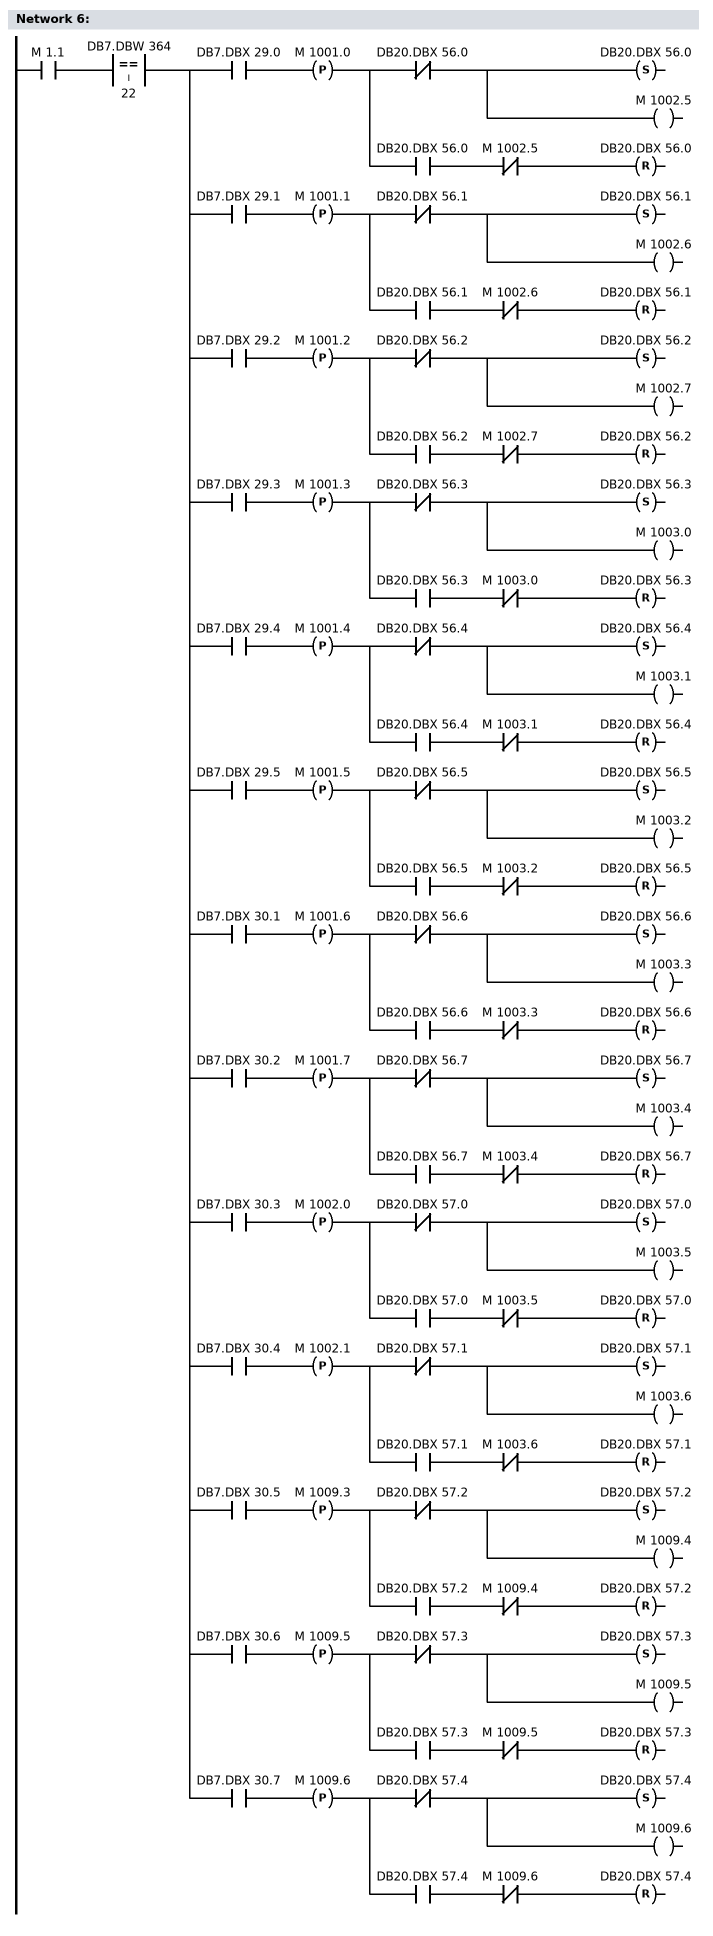
NETWORK
TITLE =
      A     M 1.1;
      A(;
      L     DB7.DBW 364;
      L     22;
      ==I;
      );
      =     L 0.0;
      A     L 0.0;
      A     DB7.DBX 29.0;
      FP    M 1001.0;
      =     L 0.1;
      A     L 0.1;
      AN    DB20.DBX 56.0;
      S     DB20.DBX 56.0;
      =     M 1002.5;
      A     L 0.1;
      A     DB20.DBX 56.0;
      AN    M 1002.5;
      R     DB20.DBX 56.0;
      A     L 0.0;
      A     DB7.DBX 29.1;
      FP    M 1001.1;
      =     L 0.1;
      A     L 0.1;
      AN    DB20.DBX 56.1;
      S     DB20.DBX 56.1;
      =     M 1002.6;
      A     L 0.1;
      A     DB20.DBX 56.1;
      AN    M 1002.6;
      R     DB20.DBX 56.1;
      A     L 0.0;
      A     DB7.DBX 29.2;
      FP    M 1001.2;
      =     L 0.1;
      A     L 0.1;
      AN    DB20.DBX 56.2;
      S     DB20.DBX 56.2;
      =     M 1002.7;
      A     L 0.1;
      A     DB20.DBX 56.2;
      AN    M 1002.7;
      R     DB20.DBX 56.2;
      A     L 0.0;
      A     DB7.DBX 29.3;
      FP    M 1001.3;
      =     L 0.1;
      A     L 0.1;
      AN    DB20.DBX 56.3;
      S     DB20.DBX 56.3;
      =     M 1003.0;
      A     L 0.1;
      A     DB20.DBX 56.3;
      AN    M 1003.0;
      R     DB20.DBX 56.3;
      A     L 0.0;
      A     DB7.DBX 29.4;
      FP    M 1001.4;
      =     L 0.1;
      A     L 0.1;
      AN    DB20.DBX 56.4;
      S     DB20.DBX 56.4;
      =     M 1003.1;
      A     L 0.1;
      A     DB20.DBX 56.4;
      AN    M 1003.1;
      R     DB20.DBX 56.4;
      A     L 0.0;
      A     DB7.DBX 29.5;
      FP    M 1001.5;
      =     L 0.1;
      A     L 0.1;
      AN    DB20.DBX 56.5;
      S     DB20.DBX 56.5;
      =     M 1003.2;
      A     L 0.1;
      A     DB20.DBX 56.5;
      AN    M 1003.2;
      R     DB20.DBX 56.5;
      A     L 0.0;
      A     DB7.DBX 30.1;
      FP    M 1001.6;
      =     L 0.1;
      A     L 0.1;
      AN    DB20.DBX 56.6;
      S     DB20.DBX 56.6;
      =     M 1003.3;
      A     L 0.1;
      A     DB20.DBX 56.6;
      AN    M 1003.3;
      R     DB20.DBX 56.6;
      A     L 0.0;
      A     DB7.DBX 30.2;
      FP    M 1001.7;
      =     L 0.1;
      A     L 0.1;
      AN    DB20.DBX 56.7;
      S     DB20.DBX 56.7;
      =     M 1003.4;
      A     L 0.1;
      A     DB20.DBX 56.7;
      AN    M 1003.4;
      R     DB20.DBX 56.7;
      A     L 0.0;
      A     DB7.DBX 30.3;
      FP    M 1002.0;
      =     L 0.1;
      A     L 0.1;
      AN    DB20.DBX 57.0;
      S     DB20.DBX 57.0;
      =     M 1003.5;
      A     L 0.1;
      A     DB20.DBX 57.0;
      AN    M 1003.5;
      R     DB20.DBX 57.0;
      A     L 0.0;
      A     DB7.DBX 30.4;
      FP    M 1002.1;
      =     L 0.1;
      A     L 0.1;
      AN    DB20.DBX 57.1;
      S     DB20.DBX 57.1;
      =     M 1003.6;
      A     L 0.1;
      A     DB20.DBX 57.1;
      AN    M 1003.6;
      R     DB20.DBX 57.1;
      A     L 0.0;
      A     DB7.DBX 30.5;
      FP    M 1009.3;
      =     L 0.1;
      A     L 0.1;
      AN    DB20.DBX 57.2;
      S     DB20.DBX 57.2;
      =     M 1009.4;
      A     L 0.1;
      A     DB20.DBX 57.2;
      AN    M 1009.4;
      R     DB20.DBX 57.2;
      A     L 0.0;
      A     DB7.DBX 30.6;
      FP    M 1009.5;
      =     L 0.1;
      A     L 0.1;
      AN    DB20.DBX 57.3;
      S     DB20.DBX 57.3;
      =     M 1009.5;
      A     L 0.1;
      A     DB20.DBX 57.3;
      AN    M 1009.5;
      R     DB20.DBX 57.3;
      A     L 0.0;
      A     DB7.DBX 30.7;
      FP    M 1009.6;
      =     L 0.1;
      A     L 0.1;
      AN    DB20.DBX 57.4;
      S     DB20.DBX 57.4;
      =     M 1009.6;
      A     L 0.1;
      A     DB20.DBX 57.4;
      AN    M 1009.6;
      R     DB20.DBX 57.4;
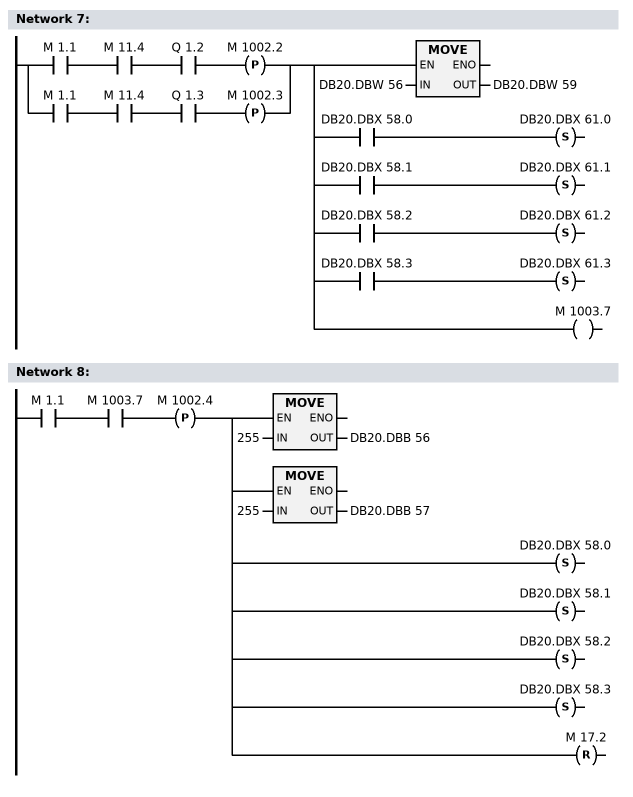
NETWORK
TITLE =
      A     M 1.1;
      A     M 11.4;
      A     Q 1.2;
      FP    M 1002.2;
      O(;
      A     M 1.1;
      A     M 11.4;
      A     Q 1.3;
      FP    M 1002.3;
      );
      =     L 0.0;
      A     L 0.0;
      JNB   M009;
      L     DB20.DBW 56;
      T     DB20.DBW 59;
M009: NOP   0;
      A     L 0.0;
      A     DB20.DBX 58.0;
      S     DB20.DBX 61.0;
      A     L 0.0;
      A     DB20.DBX 58.1;
      S     DB20.DBX 61.1;
      A     L 0.0;
      A     DB20.DBX 58.2;
      S     DB20.DBX 61.2;
      A     L 0.0;
      A     DB20.DBX 58.3;
      S     DB20.DBX 61.3;
      A     L 0.0;
      BLD   102;
      =     M 1003.7;
NETWORK
TITLE =
      A     M 1.1;
      A     M 1003.7;
      FP    M 1002.4;
      =     L 0.0;
      A     L 0.0;
      JNB   M010;
      L     255;
      T     DB20.DBB 56;
M010: NOP   0;
      A     L 0.0;
      JNB   M011;
      L     255;
      T     DB20.DBB 57;
M011: NOP   0;
      A     L 0.0;
      BLD   102;
      S     DB20.DBX 58.0;
      A     L 0.0;
      BLD   102;
      S     DB20.DBX 58.1;
      A     L 0.0;
      BLD   102;
      S     DB20.DBX 58.2;
      A     L 0.0;
      BLD   102;
      S     DB20.DBX 58.3;
      A     L 0.0;
      BLD   102;
      R     M 17.2;
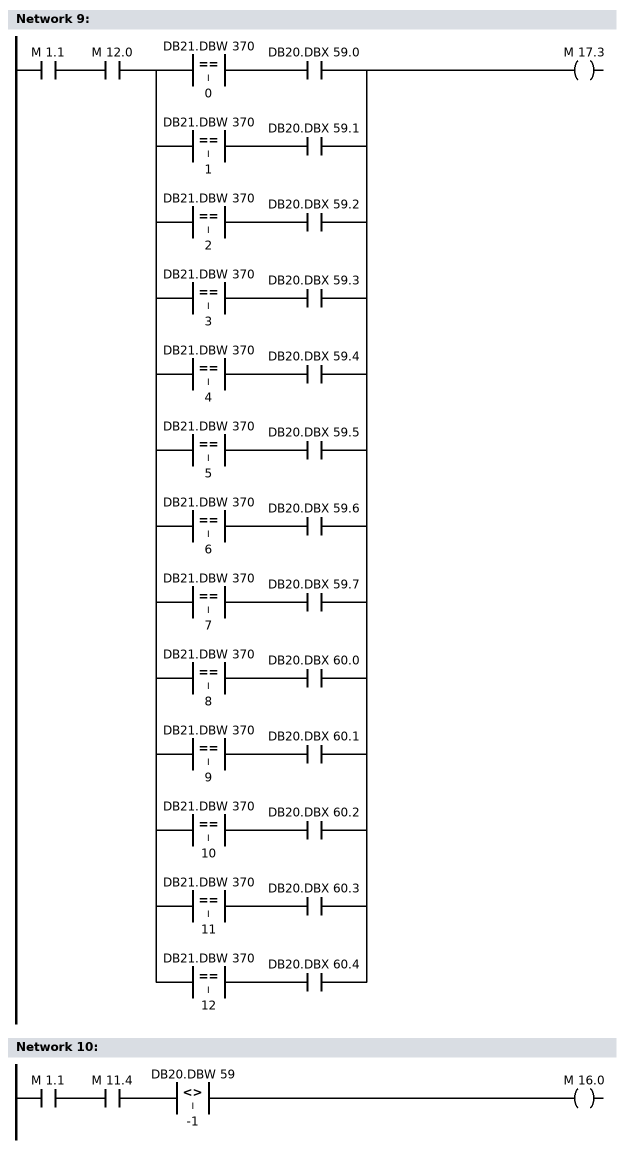
NETWORK
TITLE =
      A     M 1.1;
      A     M 12.0;
      A(;
      A(;
      L     DB21.DBW 370;
      L     0;
      ==I;
      );
      A     DB20.DBX 59.0;
      O;
      A(;
      L     DB21.DBW 370;
      L     1;
      ==I;
      );
      A     DB20.DBX 59.1;
      O;
      A(;
      L     DB21.DBW 370;
      L     2;
      ==I;
      );
      A     DB20.DBX 59.2;
      O;
      A(;
      L     DB21.DBW 370;
      L     3;
      ==I;
      );
      A     DB20.DBX 59.3;
      O;
      A(;
      L     DB21.DBW 370;
      L     4;
      ==I;
      );
      A     DB20.DBX 59.4;
      O;
      A(;
      L     DB21.DBW 370;
      L     5;
      ==I;
      );
      A     DB20.DBX 59.5;
      O;
      A(;
      L     DB21.DBW 370;
      L     6;
      ==I;
      );
      A     DB20.DBX 59.6;
      O;
      A(;
      L     DB21.DBW 370;
      L     7;
      ==I;
      );
      A     DB20.DBX 59.7;
      O;
      A(;
      L     DB21.DBW 370;
      L     8;
      ==I;
      );
      A     DB20.DBX 60.0;
      O;
      A(;
      L     DB21.DBW 370;
      L     9;
      ==I;
      );
      A     DB20.DBX 60.1;
      O;
      A(;
      L     DB21.DBW 370;
      L     10;
      ==I;
      );
      A     DB20.DBX 60.2;
      O;
      A(;
      L     DB21.DBW 370;
      L     11;
      ==I;
      );
      A     DB20.DBX 60.3;
      O;
      A(;
      L     DB21.DBW 370;
      L     12;
      ==I;
      );
      A     DB20.DBX 60.4;
      );
      =     M 17.3;
NETWORK
TITLE =
      A     M 1.1;
      A     M 11.4;
      A(;
      L     DB20.DBW 59;
      L     -1;
      <>I;
      );
      =     M 16.0;
END_FUNCTION

FUNCTION FC 54 : VOID
VERSION : 0.1
BEGIN
// (block stored without names or comments; labels and parameter names are numbered)
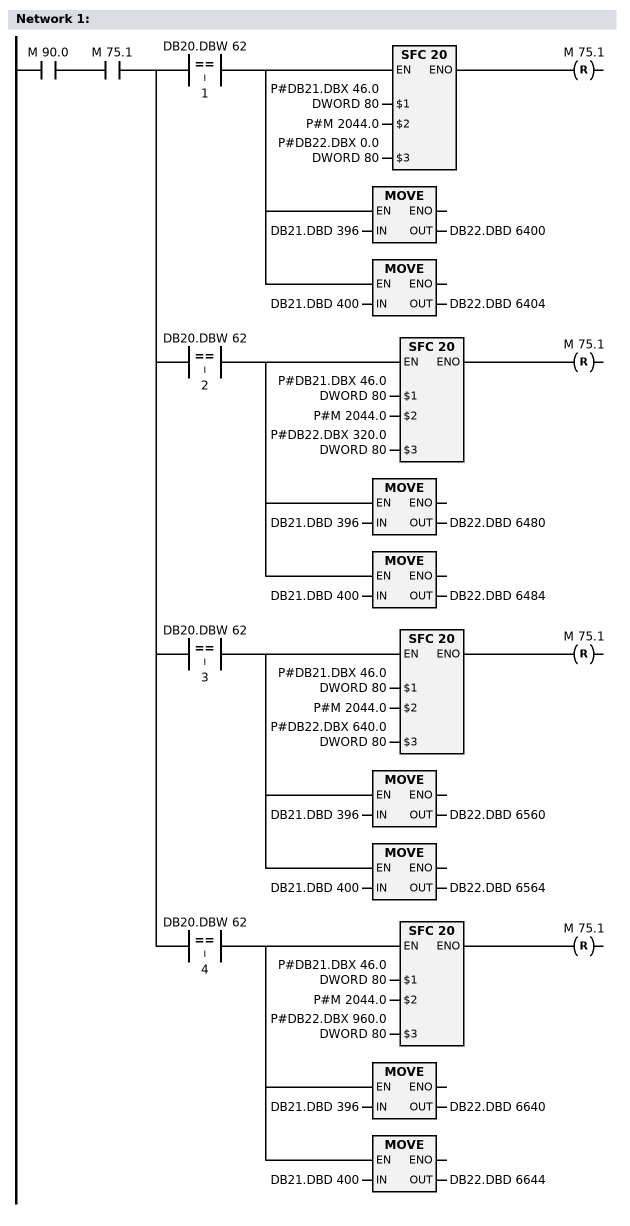
NETWORK
TITLE =
      A     M 90.0;
      A     M 75.1;
      =     L 0.0;
      A     L 0.0;
      A(;
      L     DB20.DBW 62;
      L     1;
      ==I;
      );
      =     L 0.1;
      A     L 0.1;
      JNB   M001;
      CALL  SFC 20 (
           $1                       := P#DB21.DBX 46.0 DWORD 80,
           $2                       := P#M 2044.0,
           $3                       := P#DB22.DBX 0.0 DWORD 80);
M001: A     BR;
      R     M 75.1;
      A     L 0.1;
      JNB   M002;
      L     DB21.DBD 396;
      T     DB22.DBD 6400;
M002: NOP   0;
      A     L 0.1;
      JNB   M003;
      L     DB21.DBD 400;
      T     DB22.DBD 6404;
M003: NOP   0;
      A     L 0.0;
      A(;
      L     DB20.DBW 62;
      L     2;
      ==I;
      );
      =     L 0.1;
      A     L 0.1;
      JNB   M004;
      CALL  SFC 20 (
           $1                       := P#DB21.DBX 46.0 DWORD 80,
           $2                       := P#M 2044.0,
           $3                       := P#DB22.DBX 320.0 DWORD 80);
M004: A     BR;
      R     M 75.1;
      A     L 0.1;
      JNB   M005;
      L     DB21.DBD 396;
      T     DB22.DBD 6480;
M005: NOP   0;
      A     L 0.1;
      JNB   M006;
      L     DB21.DBD 400;
      T     DB22.DBD 6484;
M006: NOP   0;
      A     L 0.0;
      A(;
      L     DB20.DBW 62;
      L     3;
      ==I;
      );
      =     L 0.1;
      A     L 0.1;
      JNB   M007;
      CALL  SFC 20 (
           $1                       := P#DB21.DBX 46.0 DWORD 80,
           $2                       := P#M 2044.0,
           $3                       := P#DB22.DBX 640.0 DWORD 80);
M007: A     BR;
      R     M 75.1;
      A     L 0.1;
      JNB   M008;
      L     DB21.DBD 396;
      T     DB22.DBD 6560;
M008: NOP   0;
      A     L 0.1;
      JNB   M009;
      L     DB21.DBD 400;
      T     DB22.DBD 6564;
M009: NOP   0;
      A     L 0.0;
      A(;
      L     DB20.DBW 62;
      L     4;
      ==I;
      );
      =     L 0.1;
      A     L 0.1;
      JNB   M010;
      CALL  SFC 20 (
           $1                       := P#DB21.DBX 46.0 DWORD 80,
           $2                       := P#M 2044.0,
           $3                       := P#DB22.DBX 960.0 DWORD 80);
M010: A     BR;
      R     M 75.1;
      A     L 0.1;
      JNB   M011;
      L     DB21.DBD 396;
      T     DB22.DBD 6640;
M011: NOP   0;
      A     L 0.1;
      JNB   M012;
      L     DB21.DBD 400;
      T     DB22.DBD 6644;
M012: NOP   0;
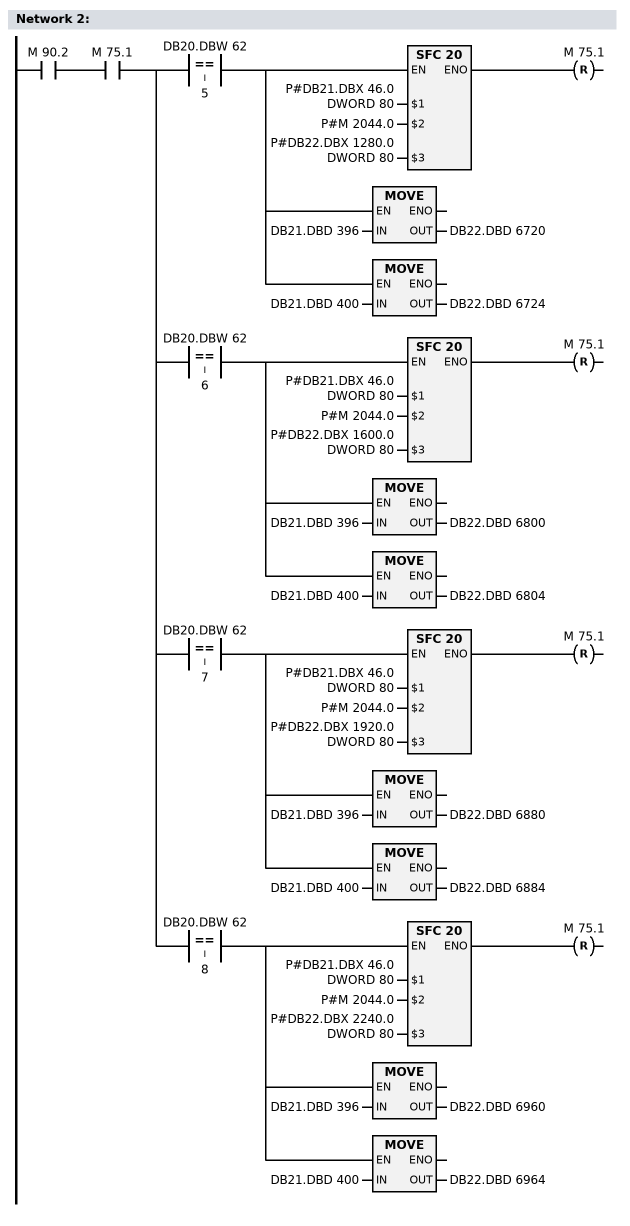
NETWORK
TITLE =
      A     M 90.2;
      A     M 75.1;
      =     L 0.0;
      A     L 0.0;
      A(;
      L     DB20.DBW 62;
      L     5;
      ==I;
      );
      =     L 0.1;
      A     L 0.1;
      JNB   M013;
      CALL  SFC 20 (
           $1                       := P#DB21.DBX 46.0 DWORD 80,
           $2                       := P#M 2044.0,
           $3                       := P#DB22.DBX 1280.0 DWORD 80);
M013: A     BR;
      R     M 75.1;
      A     L 0.1;
      JNB   M014;
      L     DB21.DBD 396;
      T     DB22.DBD 6720;
M014: NOP   0;
      A     L 0.1;
      JNB   M015;
      L     DB21.DBD 400;
      T     DB22.DBD 6724;
M015: NOP   0;
      A     L 0.0;
      A(;
      L     DB20.DBW 62;
      L     6;
      ==I;
      );
      =     L 0.1;
      A     L 0.1;
      JNB   M016;
      CALL  SFC 20 (
           $1                       := P#DB21.DBX 46.0 DWORD 80,
           $2                       := P#M 2044.0,
           $3                       := P#DB22.DBX 1600.0 DWORD 80);
M016: A     BR;
      R     M 75.1;
      A     L 0.1;
      JNB   M017;
      L     DB21.DBD 396;
      T     DB22.DBD 6800;
M017: NOP   0;
      A     L 0.1;
      JNB   M018;
      L     DB21.DBD 400;
      T     DB22.DBD 6804;
M018: NOP   0;
      A     L 0.0;
      A(;
      L     DB20.DBW 62;
      L     7;
      ==I;
      );
      =     L 0.1;
      A     L 0.1;
      JNB   M019;
      CALL  SFC 20 (
           $1                       := P#DB21.DBX 46.0 DWORD 80,
           $2                       := P#M 2044.0,
           $3                       := P#DB22.DBX 1920.0 DWORD 80);
M019: A     BR;
      R     M 75.1;
      A     L 0.1;
      JNB   M020;
      L     DB21.DBD 396;
      T     DB22.DBD 6880;
M020: NOP   0;
      A     L 0.1;
      JNB   M021;
      L     DB21.DBD 400;
      T     DB22.DBD 6884;
M021: NOP   0;
      A     L 0.0;
      A(;
      L     DB20.DBW 62;
      L     8;
      ==I;
      );
      =     L 0.1;
      A     L 0.1;
      JNB   M022;
      CALL  SFC 20 (
           $1                       := P#DB21.DBX 46.0 DWORD 80,
           $2                       := P#M 2044.0,
           $3                       := P#DB22.DBX 2240.0 DWORD 80);
M022: A     BR;
      R     M 75.1;
      A     L 0.1;
      JNB   M023;
      L     DB21.DBD 396;
      T     DB22.DBD 6960;
M023: NOP   0;
      A     L 0.1;
      JNB   M024;
      L     DB21.DBD 400;
      T     DB22.DBD 6964;
M024: NOP   0;
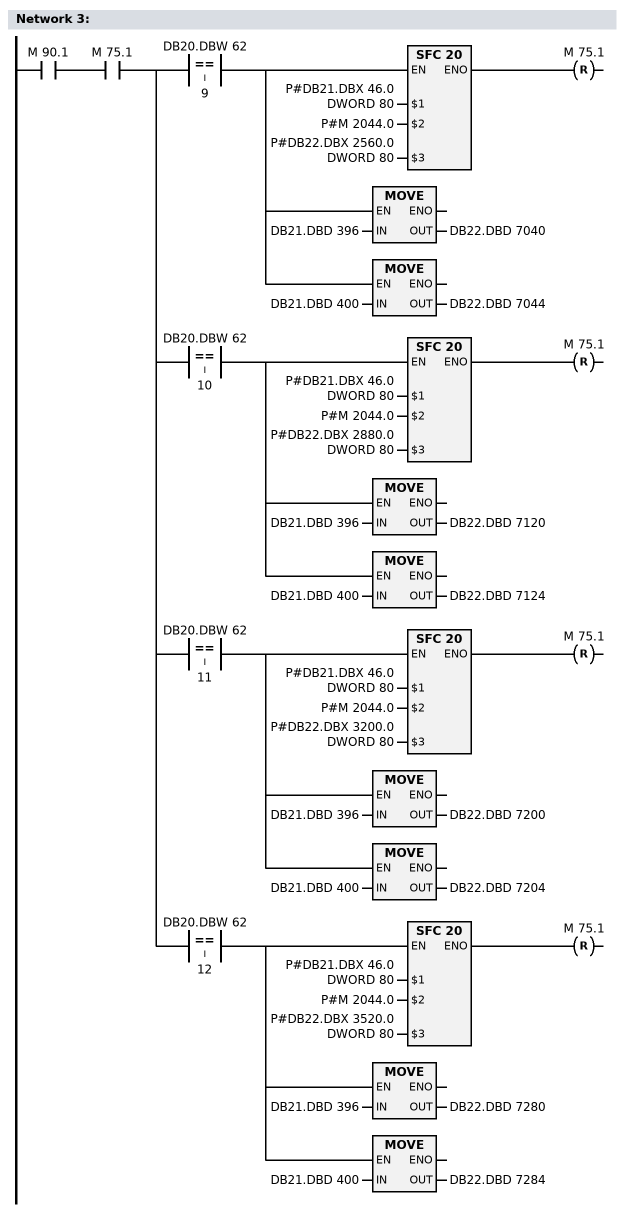
NETWORK
TITLE =
      A     M 90.1;
      A     M 75.1;
      =     L 0.0;
      A     L 0.0;
      A(;
      L     DB20.DBW 62;
      L     9;
      ==I;
      );
      =     L 0.1;
      A     L 0.1;
      JNB   M025;
      CALL  SFC 20 (
           $1                       := P#DB21.DBX 46.0 DWORD 80,
           $2                       := P#M 2044.0,
           $3                       := P#DB22.DBX 2560.0 DWORD 80);
M025: A     BR;
      R     M 75.1;
      A     L 0.1;
      JNB   M026;
      L     DB21.DBD 396;
      T     DB22.DBD 7040;
M026: NOP   0;
      A     L 0.1;
      JNB   M027;
      L     DB21.DBD 400;
      T     DB22.DBD 7044;
M027: NOP   0;
      A     L 0.0;
      A(;
      L     DB20.DBW 62;
      L     10;
      ==I;
      );
      =     L 0.1;
      A     L 0.1;
      JNB   M028;
      CALL  SFC 20 (
           $1                       := P#DB21.DBX 46.0 DWORD 80,
           $2                       := P#M 2044.0,
           $3                       := P#DB22.DBX 2880.0 DWORD 80);
M028: A     BR;
      R     M 75.1;
      A     L 0.1;
      JNB   M029;
      L     DB21.DBD 396;
      T     DB22.DBD 7120;
M029: NOP   0;
      A     L 0.1;
      JNB   M030;
      L     DB21.DBD 400;
      T     DB22.DBD 7124;
M030: NOP   0;
      A     L 0.0;
      A(;
      L     DB20.DBW 62;
      L     11;
      ==I;
      );
      =     L 0.1;
      A     L 0.1;
      JNB   M031;
      CALL  SFC 20 (
           $1                       := P#DB21.DBX 46.0 DWORD 80,
           $2                       := P#M 2044.0,
           $3                       := P#DB22.DBX 3200.0 DWORD 80);
M031: A     BR;
      R     M 75.1;
      A     L 0.1;
      JNB   M032;
      L     DB21.DBD 396;
      T     DB22.DBD 7200;
M032: NOP   0;
      A     L 0.1;
      JNB   M033;
      L     DB21.DBD 400;
      T     DB22.DBD 7204;
M033: NOP   0;
      A     L 0.0;
      A(;
      L     DB20.DBW 62;
      L     12;
      ==I;
      );
      =     L 0.1;
      A     L 0.1;
      JNB   M034;
      CALL  SFC 20 (
           $1                       := P#DB21.DBX 46.0 DWORD 80,
           $2                       := P#M 2044.0,
           $3                       := P#DB22.DBX 3520.0 DWORD 80);
M034: A     BR;
      R     M 75.1;
      A     L 0.1;
      JNB   M035;
      L     DB21.DBD 396;
      T     DB22.DBD 7280;
M035: NOP   0;
      A     L 0.1;
      JNB   M036;
      L     DB21.DBD 400;
      T     DB22.DBD 7284;
M036: NOP   0;
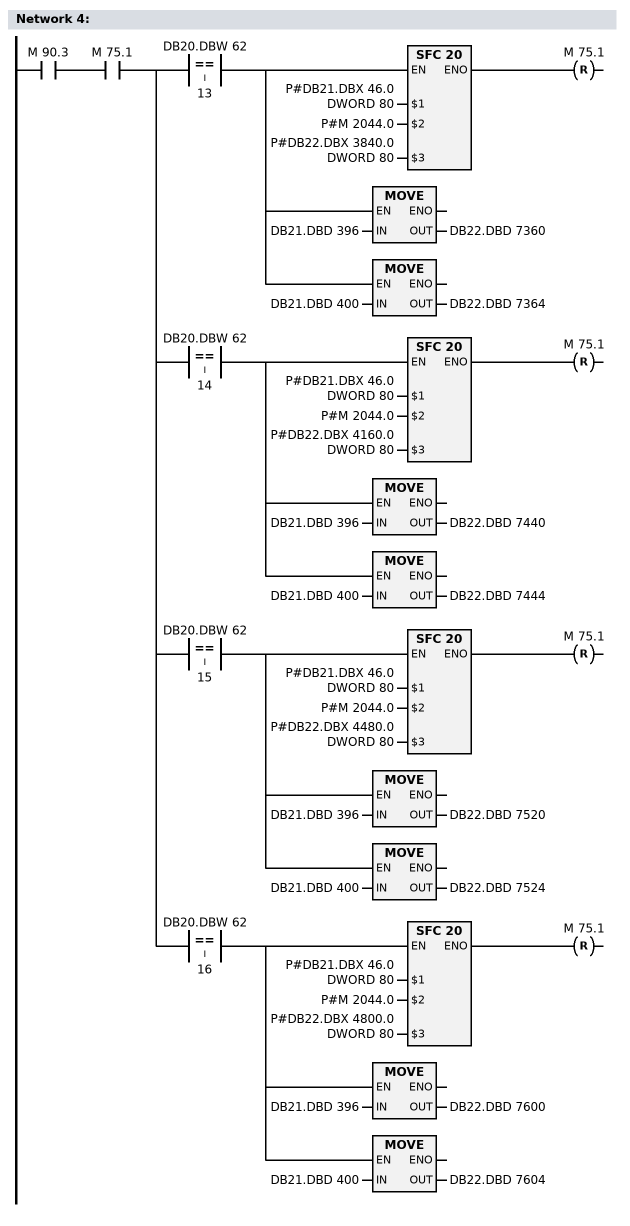
NETWORK
TITLE =
      A     M 90.3;
      A     M 75.1;
      =     L 0.0;
      A     L 0.0;
      A(;
      L     DB20.DBW 62;
      L     13;
      ==I;
      );
      =     L 0.1;
      A     L 0.1;
      JNB   M037;
      CALL  SFC 20 (
           $1                       := P#DB21.DBX 46.0 DWORD 80,
           $2                       := P#M 2044.0,
           $3                       := P#DB22.DBX 3840.0 DWORD 80);
M037: A     BR;
      R     M 75.1;
      A     L 0.1;
      JNB   M038;
      L     DB21.DBD 396;
      T     DB22.DBD 7360;
M038: NOP   0;
      A     L 0.1;
      JNB   M039;
      L     DB21.DBD 400;
      T     DB22.DBD 7364;
M039: NOP   0;
      A     L 0.0;
      A(;
      L     DB20.DBW 62;
      L     14;
      ==I;
      );
      =     L 0.1;
      A     L 0.1;
      JNB   M040;
      CALL  SFC 20 (
           $1                       := P#DB21.DBX 46.0 DWORD 80,
           $2                       := P#M 2044.0,
           $3                       := P#DB22.DBX 4160.0 DWORD 80);
M040: A     BR;
      R     M 75.1;
      A     L 0.1;
      JNB   M041;
      L     DB21.DBD 396;
      T     DB22.DBD 7440;
M041: NOP   0;
      A     L 0.1;
      JNB   M042;
      L     DB21.DBD 400;
      T     DB22.DBD 7444;
M042: NOP   0;
      A     L 0.0;
      A(;
      L     DB20.DBW 62;
      L     15;
      ==I;
      );
      =     L 0.1;
      A     L 0.1;
      JNB   M043;
      CALL  SFC 20 (
           $1                       := P#DB21.DBX 46.0 DWORD 80,
           $2                       := P#M 2044.0,
           $3                       := P#DB22.DBX 4480.0 DWORD 80);
M043: A     BR;
      R     M 75.1;
      A     L 0.1;
      JNB   M044;
      L     DB21.DBD 396;
      T     DB22.DBD 7520;
M044: NOP   0;
      A     L 0.1;
      JNB   M045;
      L     DB21.DBD 400;
      T     DB22.DBD 7524;
M045: NOP   0;
      A     L 0.0;
      A(;
      L     DB20.DBW 62;
      L     16;
      ==I;
      );
      =     L 0.1;
      A     L 0.1;
      JNB   M046;
      CALL  SFC 20 (
           $1                       := P#DB21.DBX 46.0 DWORD 80,
           $2                       := P#M 2044.0,
           $3                       := P#DB22.DBX 4800.0 DWORD 80);
M046: A     BR;
      R     M 75.1;
      A     L 0.1;
      JNB   M047;
      L     DB21.DBD 396;
      T     DB22.DBD 7600;
M047: NOP   0;
      A     L 0.1;
      JNB   M048;
      L     DB21.DBD 400;
      T     DB22.DBD 7604;
M048: NOP   0;
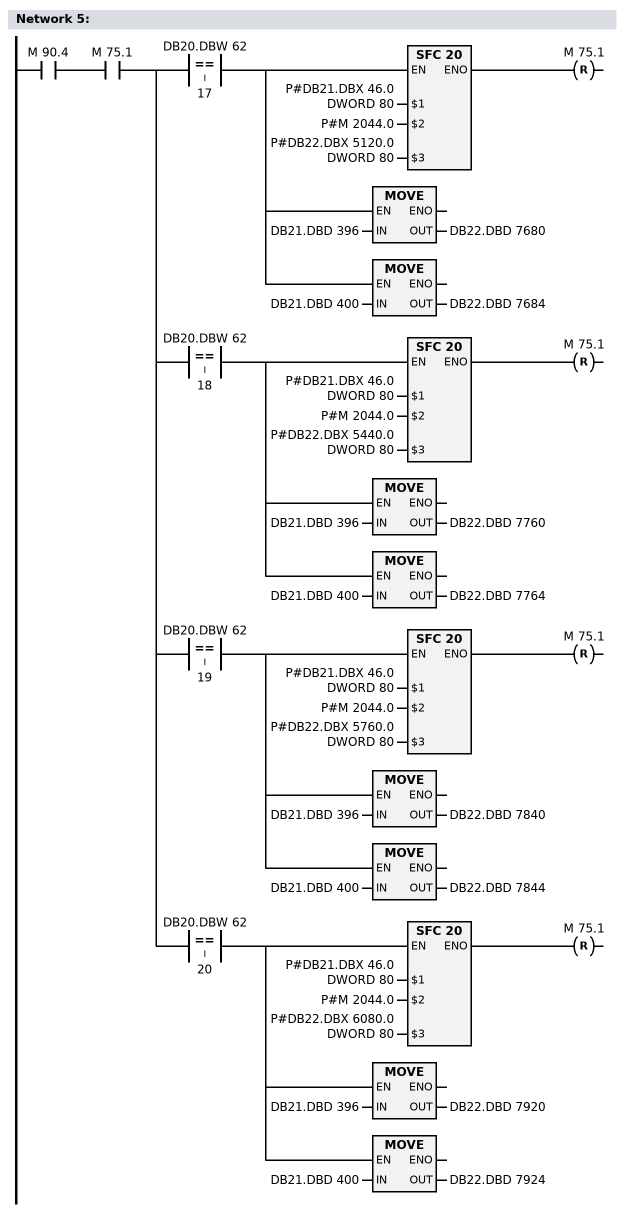
NETWORK
TITLE =
      A     M 90.4;
      A     M 75.1;
      =     L 0.0;
      A     L 0.0;
      A(;
      L     DB20.DBW 62;
      L     17;
      ==I;
      );
      =     L 0.1;
      A     L 0.1;
      JNB   M049;
      CALL  SFC 20 (
           $1                       := P#DB21.DBX 46.0 DWORD 80,
           $2                       := P#M 2044.0,
           $3                       := P#DB22.DBX 5120.0 DWORD 80);
M049: A     BR;
      R     M 75.1;
      A     L 0.1;
      JNB   M050;
      L     DB21.DBD 396;
      T     DB22.DBD 7680;
M050: NOP   0;
      A     L 0.1;
      JNB   M051;
      L     DB21.DBD 400;
      T     DB22.DBD 7684;
M051: NOP   0;
      A     L 0.0;
      A(;
      L     DB20.DBW 62;
      L     18;
      ==I;
      );
      =     L 0.1;
      A     L 0.1;
      JNB   M052;
      CALL  SFC 20 (
           $1                       := P#DB21.DBX 46.0 DWORD 80,
           $2                       := P#M 2044.0,
           $3                       := P#DB22.DBX 5440.0 DWORD 80);
M052: A     BR;
      R     M 75.1;
      A     L 0.1;
      JNB   M053;
      L     DB21.DBD 396;
      T     DB22.DBD 7760;
M053: NOP   0;
      A     L 0.1;
      JNB   M054;
      L     DB21.DBD 400;
      T     DB22.DBD 7764;
M054: NOP   0;
      A     L 0.0;
      A(;
      L     DB20.DBW 62;
      L     19;
      ==I;
      );
      =     L 0.1;
      A     L 0.1;
      JNB   M055;
      CALL  SFC 20 (
           $1                       := P#DB21.DBX 46.0 DWORD 80,
           $2                       := P#M 2044.0,
           $3                       := P#DB22.DBX 5760.0 DWORD 80);
M055: A     BR;
      R     M 75.1;
      A     L 0.1;
      JNB   M056;
      L     DB21.DBD 396;
      T     DB22.DBD 7840;
M056: NOP   0;
      A     L 0.1;
      JNB   M057;
      L     DB21.DBD 400;
      T     DB22.DBD 7844;
M057: NOP   0;
      A     L 0.0;
      A(;
      L     DB20.DBW 62;
      L     20;
      ==I;
      );
      =     L 0.1;
      A     L 0.1;
      JNB   M058;
      CALL  SFC 20 (
           $1                       := P#DB21.DBX 46.0 DWORD 80,
           $2                       := P#M 2044.0,
           $3                       := P#DB22.DBX 6080.0 DWORD 80);
M058: A     BR;
      R     M 75.1;
      A     L 0.1;
      JNB   M059;
      L     DB21.DBD 396;
      T     DB22.DBD 7920;
M059: NOP   0;
      A     L 0.1;
      JNB   M060;
      L     DB21.DBD 400;
      T     DB22.DBD 7924;
M060: NOP   0;
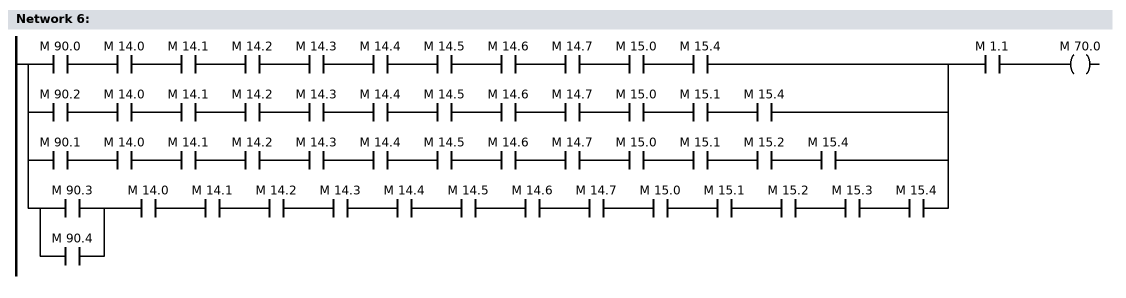
NETWORK
TITLE =
      A(;
      A     M 90.0;
      A     M 14.0;
      A     M 14.1;
      A     M 14.2;
      A     M 14.3;
      A     M 14.4;
      A     M 14.5;
      A     M 14.6;
      A     M 14.7;
      A     M 15.0;
      A     M 15.4;
      O;
      A     M 90.2;
      A     M 14.0;
      A     M 14.1;
      A     M 14.2;
      A     M 14.3;
      A     M 14.4;
      A     M 14.5;
      A     M 14.6;
      A     M 14.7;
      A     M 15.0;
      A     M 15.1;
      A     M 15.4;
      O;
      A     M 90.1;
      A     M 14.0;
      A     M 14.1;
      A     M 14.2;
      A     M 14.3;
      A     M 14.4;
      A     M 14.5;
      A     M 14.6;
      A     M 14.7;
      A     M 15.0;
      A     M 15.1;
      A     M 15.2;
      A     M 15.4;
      O;
      A(;
      O     M 90.3;
      O     M 90.4;
      );
      A     M 14.0;
      A     M 14.1;
      A     M 14.2;
      A     M 14.3;
      A     M 14.4;
      A     M 14.5;
      A     M 14.6;
      A     M 14.7;
      A     M 15.0;
      A     M 15.1;
      A     M 15.2;
      A     M 15.3;
      A     M 15.4;
      );
      A     M 1.1;
      =     M 70.0;
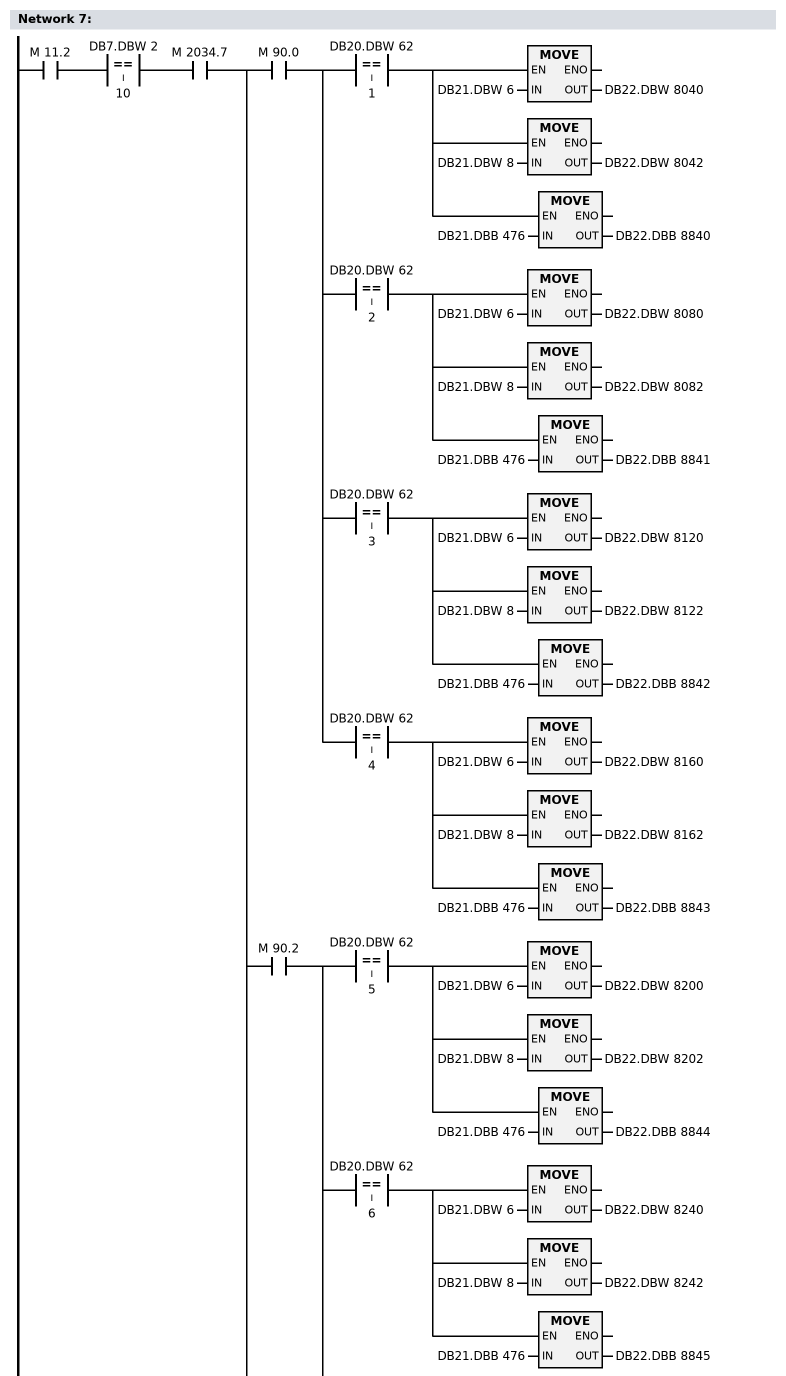
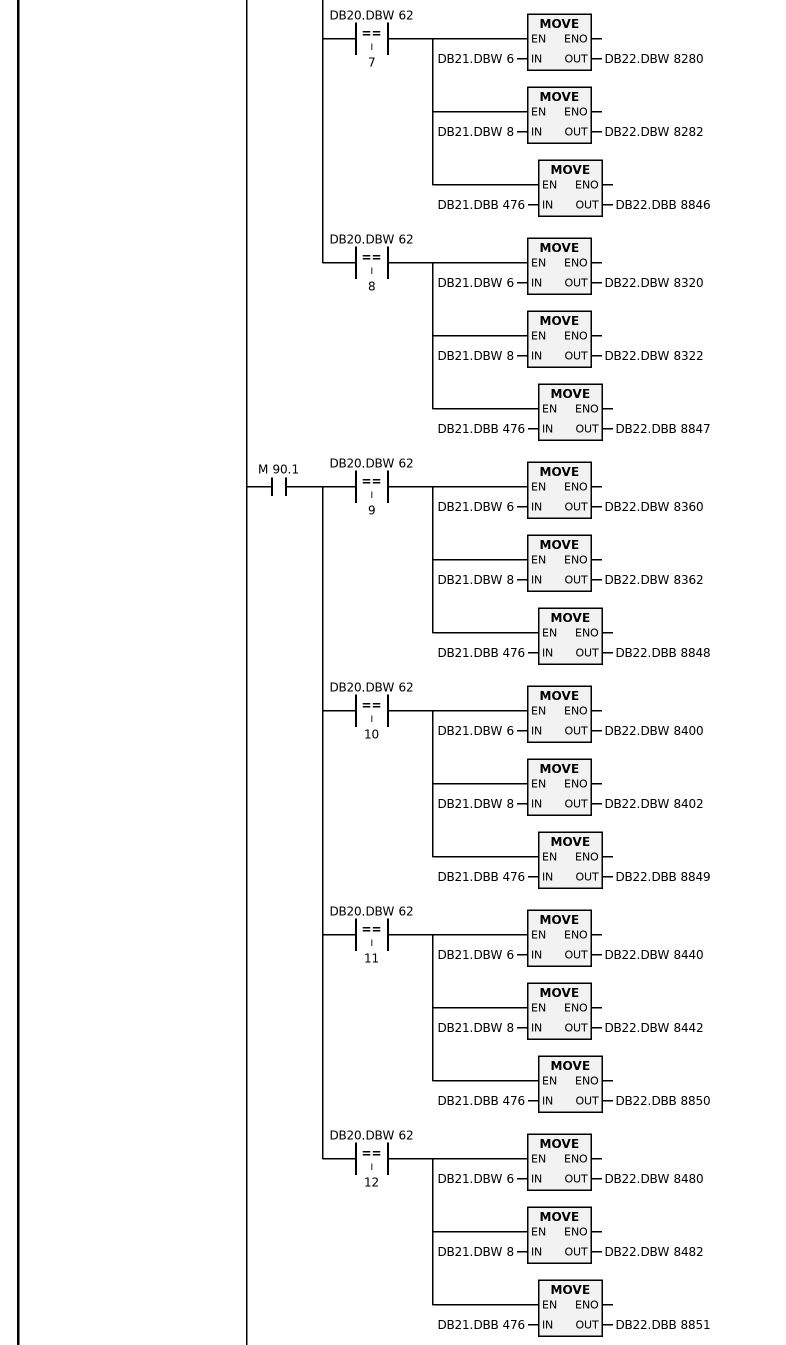
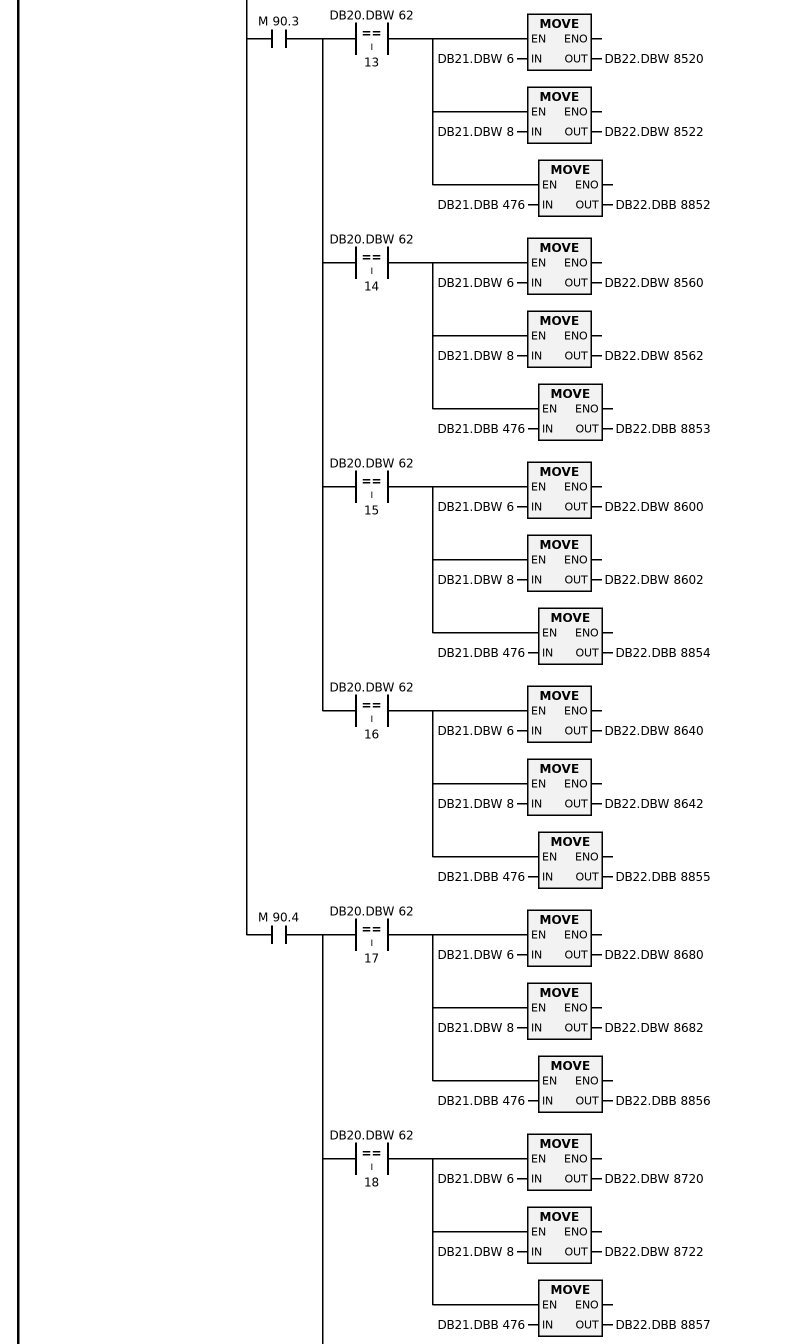
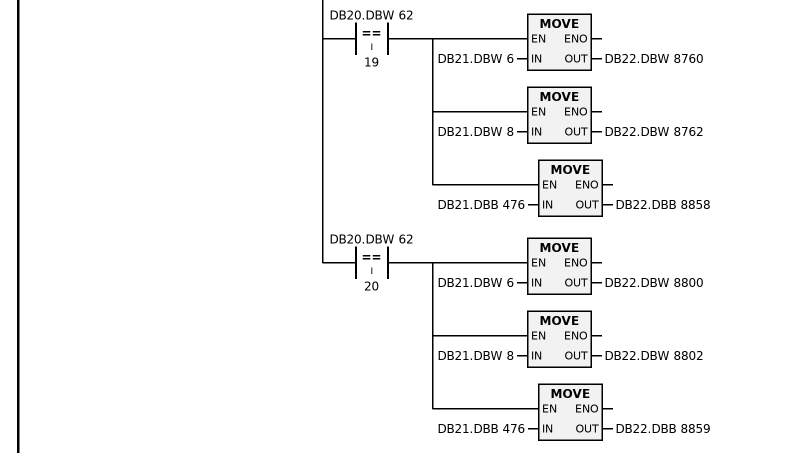
NETWORK
TITLE =
      A     M 11.2;
      A(;
      L     DB7.DBW 2;
      L     10;
      ==I;
      );
      A     M 2034.7;
      =     L 0.0;
      A     L 0.0;
      A     M 90.0;
      =     L 0.1;
      A     L 0.1;
      A(;
      L     DB20.DBW 62;
      L     1;
      ==I;
      );
      =     L 0.2;
      A     L 0.2;
      JNB   M061;
      L     DB21.DBW 6;
      T     DB22.DBW 8040;
M061: NOP   0;
      A     L 0.2;
      JNB   M062;
      L     DB21.DBW 8;
      T     DB22.DBW 8042;
M062: NOP   0;
      A     L 0.2;
      JNB   M063;
      L     DB21.DBB 476;
      T     DB22.DBB 8840;
M063: NOP   0;
      A     L 0.1;
      A(;
      L     DB20.DBW 62;
      L     2;
      ==I;
      );
      =     L 0.2;
      A     L 0.2;
      JNB   M064;
      L     DB21.DBW 6;
      T     DB22.DBW 8080;
M064: NOP   0;
      A     L 0.2;
      JNB   M065;
      L     DB21.DBW 8;
      T     DB22.DBW 8082;
M065: NOP   0;
      A     L 0.2;
      JNB   M066;
      L     DB21.DBB 476;
      T     DB22.DBB 8841;
M066: NOP   0;
      A     L 0.1;
      A(;
      L     DB20.DBW 62;
      L     3;
      ==I;
      );
      =     L 0.2;
      A     L 0.2;
      JNB   M067;
      L     DB21.DBW 6;
      T     DB22.DBW 8120;
M067: NOP   0;
      A     L 0.2;
      JNB   M068;
      L     DB21.DBW 8;
      T     DB22.DBW 8122;
M068: NOP   0;
      A     L 0.2;
      JNB   M069;
      L     DB21.DBB 476;
      T     DB22.DBB 8842;
M069: NOP   0;
      A     L 0.1;
      A(;
      L     DB20.DBW 62;
      L     4;
      ==I;
      );
      =     L 0.2;
      A     L 0.2;
      JNB   M070;
      L     DB21.DBW 6;
      T     DB22.DBW 8160;
M070: NOP   0;
      A     L 0.2;
      JNB   M071;
      L     DB21.DBW 8;
      T     DB22.DBW 8162;
M071: NOP   0;
      A     L 0.2;
      JNB   M072;
      L     DB21.DBB 476;
      T     DB22.DBB 8843;
M072: NOP   0;
      A     L 0.0;
      A     M 90.2;
      =     L 0.1;
      A     L 0.1;
      A(;
      L     DB20.DBW 62;
      L     5;
      ==I;
      );
      =     L 0.2;
      A     L 0.2;
      JNB   M073;
      L     DB21.DBW 6;
      T     DB22.DBW 8200;
M073: NOP   0;
      A     L 0.2;
      JNB   M074;
      L     DB21.DBW 8;
      T     DB22.DBW 8202;
M074: NOP   0;
      A     L 0.2;
      JNB   M075;
      L     DB21.DBB 476;
      T     DB22.DBB 8844;
M075: NOP   0;
      A     L 0.1;
      A(;
      L     DB20.DBW 62;
      L     6;
      ==I;
      );
      =     L 0.2;
      A     L 0.2;
      JNB   M076;
      L     DB21.DBW 6;
      T     DB22.DBW 8240;
M076: NOP   0;
      A     L 0.2;
      JNB   M077;
      L     DB21.DBW 8;
      T     DB22.DBW 8242;
M077: NOP   0;
      A     L 0.2;
      JNB   M078;
      L     DB21.DBB 476;
      T     DB22.DBB 8845;
M078: NOP   0;
      A     L 0.1;
      A(;
      L     DB20.DBW 62;
      L     7;
      ==I;
      );
      =     L 0.2;
      A     L 0.2;
      JNB   M079;
      L     DB21.DBW 6;
      T     DB22.DBW 8280;
M079: NOP   0;
      A     L 0.2;
      JNB   M080;
      L     DB21.DBW 8;
      T     DB22.DBW 8282;
M080: NOP   0;
      A     L 0.2;
      JNB   M081;
      L     DB21.DBB 476;
      T     DB22.DBB 8846;
M081: NOP   0;
      A     L 0.1;
      A(;
      L     DB20.DBW 62;
      L     8;
      ==I;
      );
      =     L 0.2;
      A     L 0.2;
      JNB   M082;
      L     DB21.DBW 6;
      T     DB22.DBW 8320;
M082: NOP   0;
      A     L 0.2;
      JNB   M083;
      L     DB21.DBW 8;
      T     DB22.DBW 8322;
M083: NOP   0;
      A     L 0.2;
      JNB   M084;
      L     DB21.DBB 476;
      T     DB22.DBB 8847;
M084: NOP   0;
      A     L 0.0;
      A     M 90.1;
      =     L 0.1;
      A     L 0.1;
      A(;
      L     DB20.DBW 62;
      L     9;
      ==I;
      );
      =     L 0.2;
      A     L 0.2;
      JNB   M085;
      L     DB21.DBW 6;
      T     DB22.DBW 8360;
M085: NOP   0;
      A     L 0.2;
      JNB   M086;
      L     DB21.DBW 8;
      T     DB22.DBW 8362;
M086: NOP   0;
      A     L 0.2;
      JNB   M087;
      L     DB21.DBB 476;
      T     DB22.DBB 8848;
M087: NOP   0;
      A     L 0.1;
      A(;
      L     DB20.DBW 62;
      L     10;
      ==I;
      );
      =     L 0.2;
      A     L 0.2;
      JNB   M088;
      L     DB21.DBW 6;
      T     DB22.DBW 8400;
M088: NOP   0;
      A     L 0.2;
      JNB   M089;
      L     DB21.DBW 8;
      T     DB22.DBW 8402;
M089: NOP   0;
      A     L 0.2;
      JNB   M090;
      L     DB21.DBB 476;
      T     DB22.DBB 8849;
M090: NOP   0;
      A     L 0.1;
      A(;
      L     DB20.DBW 62;
      L     11;
      ==I;
      );
      =     L 0.2;
      A     L 0.2;
      JNB   M091;
      L     DB21.DBW 6;
      T     DB22.DBW 8440;
M091: NOP   0;
      A     L 0.2;
      JNB   M092;
      L     DB21.DBW 8;
      T     DB22.DBW 8442;
M092: NOP   0;
      A     L 0.2;
      JNB   M093;
      L     DB21.DBB 476;
      T     DB22.DBB 8850;
M093: NOP   0;
      A     L 0.1;
      A(;
      L     DB20.DBW 62;
      L     12;
      ==I;
      );
      =     L 0.2;
      A     L 0.2;
      JNB   M094;
      L     DB21.DBW 6;
      T     DB22.DBW 8480;
M094: NOP   0;
      A     L 0.2;
      JNB   M095;
      L     DB21.DBW 8;
      T     DB22.DBW 8482;
M095: NOP   0;
      A     L 0.2;
      JNB   M096;
      L     DB21.DBB 476;
      T     DB22.DBB 8851;
M096: NOP   0;
      A     L 0.0;
      A     M 90.3;
      =     L 0.1;
      A     L 0.1;
      A(;
      L     DB20.DBW 62;
      L     13;
      ==I;
      );
      =     L 0.2;
      A     L 0.2;
      JNB   M097;
      L     DB21.DBW 6;
      T     DB22.DBW 8520;
M097: NOP   0;
      A     L 0.2;
      JNB   M098;
      L     DB21.DBW 8;
      T     DB22.DBW 8522;
M098: NOP   0;
      A     L 0.2;
      JNB   M099;
      L     DB21.DBB 476;
      T     DB22.DBB 8852;
M099: NOP   0;
      A     L 0.1;
      A(;
      L     DB20.DBW 62;
      L     14;
      ==I;
      );
      =     L 0.2;
      A     L 0.2;
      JNB   M100;
      L     DB21.DBW 6;
      T     DB22.DBW 8560;
M100: NOP   0;
      A     L 0.2;
      JNB   M101;
      L     DB21.DBW 8;
      T     DB22.DBW 8562;
M101: NOP   0;
      A     L 0.2;
      JNB   M102;
      L     DB21.DBB 476;
      T     DB22.DBB 8853;
M102: NOP   0;
      A     L 0.1;
      A(;
      L     DB20.DBW 62;
      L     15;
      ==I;
      );
      =     L 0.2;
      A     L 0.2;
      JNB   M103;
      L     DB21.DBW 6;
      T     DB22.DBW 8600;
M103: NOP   0;
      A     L 0.2;
      JNB   M104;
      L     DB21.DBW 8;
      T     DB22.DBW 8602;
M104: NOP   0;
      A     L 0.2;
      JNB   M105;
      L     DB21.DBB 476;
      T     DB22.DBB 8854;
M105: NOP   0;
      A     L 0.1;
      A(;
      L     DB20.DBW 62;
      L     16;
      ==I;
      );
      =     L 0.2;
      A     L 0.2;
      JNB   M106;
      L     DB21.DBW 6;
      T     DB22.DBW 8640;
M106: NOP   0;
      A     L 0.2;
      JNB   M107;
      L     DB21.DBW 8;
      T     DB22.DBW 8642;
M107: NOP   0;
      A     L 0.2;
      JNB   M108;
      L     DB21.DBB 476;
      T     DB22.DBB 8855;
M108: NOP   0;
      A     L 0.0;
      A     M 90.4;
      =     L 0.1;
      A     L 0.1;
      A(;
      L     DB20.DBW 62;
      L     17;
      ==I;
      );
      =     L 0.2;
      A     L 0.2;
      JNB   M109;
      L     DB21.DBW 6;
      T     DB22.DBW 8680;
M109: NOP   0;
      A     L 0.2;
      JNB   M110;
      L     DB21.DBW 8;
      T     DB22.DBW 8682;
M110: NOP   0;
      A     L 0.2;
      JNB   M111;
      L     DB21.DBB 476;
      T     DB22.DBB 8856;
M111: NOP   0;
      A     L 0.1;
      A(;
      L     DB20.DBW 62;
      L     18;
      ==I;
      );
      =     L 0.2;
      A     L 0.2;
      JNB   M112;
      L     DB21.DBW 6;
      T     DB22.DBW 8720;
M112: NOP   0;
      A     L 0.2;
      JNB   M113;
      L     DB21.DBW 8;
      T     DB22.DBW 8722;
M113: NOP   0;
      A     L 0.2;
      JNB   M114;
      L     DB21.DBB 476;
      T     DB22.DBB 8857;
M114: NOP   0;
      A     L 0.1;
      A(;
      L     DB20.DBW 62;
      L     19;
      ==I;
      );
      =     L 0.2;
      A     L 0.2;
      JNB   M115;
      L     DB21.DBW 6;
      T     DB22.DBW 8760;
M115: NOP   0;
      A     L 0.2;
      JNB   M116;
      L     DB21.DBW 8;
      T     DB22.DBW 8762;
M116: NOP   0;
      A     L 0.2;
      JNB   M117;
      L     DB21.DBB 476;
      T     DB22.DBB 8858;
M117: NOP   0;
      A     L 0.1;
      A(;
      L     DB20.DBW 62;
      L     20;
      ==I;
      );
      =     L 0.2;
      A     L 0.2;
      JNB   M118;
      L     DB21.DBW 6;
      T     DB22.DBW 8800;
M118: NOP   0;
      A     L 0.2;
      JNB   M119;
      L     DB21.DBW 8;
      T     DB22.DBW 8802;
M119: NOP   0;
      A     L 0.2;
      JNB   M120;
      L     DB21.DBB 476;
      T     DB22.DBB 8859;
M120: NOP   0;
NETWORK
TITLE =
NETWORK
TITLE =
      A     M 1.1;
      =     L 0.0;
      A     L 0.0;
      A(;
      A(;
      L     DB21.DBW 370;
      L     0;
      ==I;
      );
      A     M 11.4;
      O;
      A     M 11.2;
      A(;
      L     DB7.DBB 375;
      L     1;
      ==I;
      );
      A(;
      O(;
      L     DB7.DBW 2;
      L     5;
      ==I;
      );
      O(;
      L     DB7.DBW 2;
      L     11;
      ==I;
      );
      );
      );
      =     L 0.1;
      A(;
      A     L 0.1;
      A     DB21.DBX 394.0;
      JNB   M121;
      L     DB21.DBD 46;
      T     MD 588;
      SET;
      SAVE;
      CLR;
M121: A     BR;
      );
      JNB   M122;
      L     DB21.DBD 50;
      T     MD 592;
M122: NOP   0;
      A(;
      A     L 0.1;
      AN    DB21.DBX 394.0;
      JNB   M123;
      L     DB21.DBD 54;
      T     MD 588;
      SET;
      SAVE;
      CLR;
M123: A     BR;
      );
      JNB   M124;
      L     DB21.DBD 58;
      T     MD 592;
M124: NOP   0;
      A     L 0.0;
      A(;
      A(;
      L     DB21.DBW 370;
      L     1;
      ==I;
      );
      A     M 11.4;
      O;
      A     M 11.2;
      A(;
      L     DB7.DBB 375;
      L     2;
      ==I;
      );
      A(;
      O(;
      L     DB7.DBW 2;
      L     5;
      ==I;
      );
      O(;
      L     DB7.DBW 2;
      L     11;
      ==I;
      );
      );
      );
      =     L 0.1;
      A(;
      A     L 0.1;
      A     DB21.DBX 394.0;
      JNB   M125;
      L     DB21.DBD 62;
      T     MD 588;
      SET;
      SAVE;
      CLR;
M125: A     BR;
      );
      JNB   M126;
      L     DB21.DBD 66;
      T     MD 592;
M126: NOP   0;
      A(;
      A     L 0.1;
      AN    DB21.DBX 394.0;
      JNB   M127;
      L     DB21.DBD 70;
      T     MD 588;
      SET;
      SAVE;
      CLR;
M127: A     BR;
      );
      JNB   M128;
      L     DB21.DBD 74;
      T     MD 592;
M128: NOP   0;
      A     L 0.0;
      A(;
      A(;
      L     DB21.DBW 370;
      L     2;
      ==I;
      );
      A     M 11.4;
      O;
      A     M 11.2;
      A(;
      L     DB7.DBB 375;
      L     3;
      ==I;
      );
      A(;
      O(;
      L     DB7.DBW 2;
      L     5;
      ==I;
      );
      O(;
      L     DB7.DBW 2;
      L     11;
      ==I;
      );
      );
      );
      =     L 0.1;
      A(;
      A     L 0.1;
      A     DB21.DBX 394.0;
      JNB   M129;
      L     DB21.DBD 78;
      T     MD 588;
      SET;
      SAVE;
      CLR;
M129: A     BR;
      );
      JNB   M130;
      L     DB21.DBD 82;
      T     MD 592;
M130: NOP   0;
      A(;
      A     L 0.1;
      AN    DB21.DBX 394.0;
      JNB   M131;
      L     DB21.DBD 86;
      T     MD 588;
      SET;
      SAVE;
      CLR;
M131: A     BR;
      );
      JNB   M132;
      L     DB21.DBD 90;
      T     MD 592;
M132: NOP   0;
      A     L 0.0;
      A(;
      A(;
      L     DB21.DBW 370;
      L     3;
      ==I;
      );
      A     M 11.4;
      O;
      A     M 11.2;
      A(;
      L     DB7.DBB 375;
      L     4;
      ==I;
      );
      A(;
      O(;
      L     DB7.DBW 2;
      L     5;
      ==I;
      );
      O(;
      L     DB7.DBW 2;
      L     11;
      ==I;
      );
      );
      );
      =     L 0.1;
      A(;
      A     L 0.1;
      A     DB21.DBX 394.0;
      JNB   M133;
      L     DB21.DBD 94;
      T     MD 588;
      SET;
      SAVE;
      CLR;
M133: A     BR;
      );
      JNB   M134;
      L     DB21.DBD 98;
      T     MD 592;
M134: NOP   0;
      A(;
      A     L 0.1;
      AN    DB21.DBX 394.0;
      JNB   M135;
      L     DB21.DBD 102;
      T     MD 588;
      SET;
      SAVE;
      CLR;
M135: A     BR;
      );
      JNB   M136;
      L     DB21.DBD 106;
      T     MD 592;
M136: NOP   0;
      A     L 0.0;
      A(;
      A(;
      L     DB21.DBW 370;
      L     4;
      ==I;
      );
      A     M 11.4;
      O;
      A     M 11.2;
      A(;
      L     DB7.DBB 375;
      L     5;
      ==I;
      );
      A(;
      O(;
      L     DB7.DBW 2;
      L     5;
      ==I;
      );
      O(;
      L     DB7.DBW 2;
      L     11;
      ==I;
      );
      );
      );
      =     L 0.1;
      A(;
      A     L 0.1;
      A     DB21.DBX 394.0;
      JNB   M137;
      L     DB21.DBD 110;
      T     MD 588;
      SET;
      SAVE;
      CLR;
M137: A     BR;
      );
      JNB   M138;
      L     DB21.DBD 114;
      T     MD 592;
M138: NOP   0;
      A(;
      A     L 0.1;
      AN    DB21.DBX 394.0;
      JNB   M139;
      L     DB21.DBD 118;
      T     MD 588;
      SET;
      SAVE;
      CLR;
M139: A     BR;
      );
      JNB   M140;
      L     DB21.DBD 122;
      T     MD 592;
M140: NOP   0;
      A     L 0.0;
      A(;
      A(;
      L     DB21.DBW 370;
      L     5;
      ==I;
      );
      A     M 11.4;
      O;
      A     M 11.2;
      A(;
      L     DB7.DBB 375;
      L     6;
      ==I;
      );
      A(;
      O(;
      L     DB7.DBW 2;
      L     5;
      ==I;
      );
      O(;
      L     DB7.DBW 2;
      L     11;
      ==I;
      );
      );
      );
      =     L 0.1;
      A(;
      A     L 0.1;
      A     DB21.DBX 394.0;
      JNB   M141;
      L     DB21.DBD 126;
      T     MD 588;
      SET;
      SAVE;
      CLR;
M141: A     BR;
      );
      JNB   M142;
      L     DB21.DBD 130;
      T     MD 592;
M142: NOP   0;
      A(;
      A     L 0.1;
      AN    DB21.DBX 394.0;
      JNB   M143;
      L     DB21.DBD 134;
      T     MD 588;
      SET;
      SAVE;
      CLR;
M143: A     BR;
      );
      JNB   M144;
      L     DB21.DBD 138;
      T     MD 592;
M144: NOP   0;
      A     L 0.0;
      A(;
      A(;
      L     DB21.DBW 370;
      L     6;
      ==I;
      );
      A     M 11.4;
      O;
      A     M 11.2;
      A(;
      L     DB7.DBB 375;
      L     7;
      ==I;
      );
      A(;
      O(;
      L     DB7.DBW 2;
      L     5;
      ==I;
      );
      O(;
      L     DB7.DBW 2;
      L     11;
      ==I;
      );
      );
      );
      =     L 0.1;
      A(;
      A     L 0.1;
      A     DB21.DBX 394.0;
      JNB   M145;
      L     DB21.DBD 142;
      T     MD 588;
      SET;
      SAVE;
      CLR;
M145: A     BR;
      );
      JNB   M146;
      L     DB21.DBD 146;
      T     MD 592;
M146: NOP   0;
      A(;
      A     L 0.1;
      AN    DB21.DBX 394.0;
      JNB   M147;
      L     DB21.DBD 150;
      T     MD 588;
      SET;
      SAVE;
      CLR;
M147: A     BR;
      );
      JNB   M148;
      L     DB21.DBD 154;
      T     MD 592;
M148: NOP   0;
      A     L 0.0;
      A(;
      A(;
      L     DB21.DBW 370;
      L     7;
      ==I;
      );
      A     M 11.4;
      O;
      A     M 11.2;
      A(;
      L     DB7.DBB 375;
      L     8;
      ==I;
      );
      A(;
      O(;
      L     DB7.DBW 2;
      L     5;
      ==I;
      );
      O(;
      L     DB7.DBW 2;
      L     11;
      ==I;
      );
      );
      );
      =     L 0.1;
      A(;
      A     L 0.1;
      A     DB21.DBX 394.0;
      JNB   M149;
      L     DB21.DBD 158;
      T     MD 588;
      SET;
      SAVE;
      CLR;
M149: A     BR;
      );
      JNB   M150;
      L     DB21.DBD 162;
      T     MD 592;
M150: NOP   0;
      A(;
      A     L 0.1;
      AN    DB21.DBX 394.0;
      JNB   M151;
      L     DB21.DBD 166;
      T     MD 588;
      SET;
      SAVE;
      CLR;
M151: A     BR;
      );
      JNB   M152;
      L     DB21.DBD 170;
      T     MD 592;
M152: NOP   0;
      A     L 0.0;
      A(;
      A(;
      L     DB21.DBW 370;
      L     8;
      ==I;
      );
      A     M 11.4;
      O;
      A     M 11.2;
      A(;
      L     DB7.DBB 375;
      L     9;
      ==I;
      );
      A(;
      O(;
      L     DB7.DBW 2;
      L     5;
      ==I;
      );
      O(;
      L     DB7.DBW 2;
      L     11;
      ==I;
      );
      );
      );
      =     L 0.1;
      A(;
      A     L 0.1;
      A     DB21.DBX 394.0;
      JNB   M153;
      L     DB21.DBD 174;
      T     MD 588;
      SET;
      SAVE;
      CLR;
M153: A     BR;
      );
      JNB   M154;
      L     DB21.DBD 178;
      T     MD 592;
M154: NOP   0;
      A(;
      A     L 0.1;
      AN    DB21.DBX 394.0;
      JNB   M155;
      L     DB21.DBD 182;
      T     MD 588;
      SET;
      SAVE;
      CLR;
M155: A     BR;
      );
      JNB   M156;
      L     DB21.DBD 186;
      T     MD 592;
M156: NOP   0;
      A     L 0.0;
      A(;
      A(;
      L     DB21.DBW 370;
      L     9;
      ==I;
      );
      A     M 11.4;
      O;
      A     M 11.2;
      A(;
      L     DB7.DBB 375;
      L     10;
      ==I;
      );
      A(;
      O(;
      L     DB7.DBW 2;
      L     5;
      ==I;
      );
      O(;
      L     DB7.DBW 2;
      L     11;
      ==I;
      );
      );
      );
      =     L 0.1;
      A(;
      A     L 0.1;
      A     DB21.DBX 394.0;
      JNB   M157;
      L     DB21.DBD 190;
      T     MD 588;
      SET;
      SAVE;
      CLR;
M157: A     BR;
      );
      JNB   M158;
      L     DB21.DBD 194;
      T     MD 592;
M158: NOP   0;
      A(;
      A     L 0.1;
      AN    DB21.DBX 394.0;
      JNB   M159;
      L     DB21.DBD 198;
      T     MD 588;
      SET;
      SAVE;
      CLR;
M159: A     BR;
      );
      JNB   M160;
      L     DB21.DBD 202;
      T     MD 592;
M160: NOP   0;
      A     L 0.0;
      A(;
      A(;
      L     DB21.DBW 370;
      L     10;
      ==I;
      );
      A     M 11.4;
      O;
      A     M 11.2;
      A(;
      L     DB7.DBB 375;
      L     11;
      ==I;
      );
      A(;
      O(;
      L     DB7.DBW 2;
      L     5;
      ==I;
      );
      O(;
      L     DB7.DBW 2;
      L     11;
      ==I;
      );
      );
      );
      =     L 0.1;
      A(;
      A     L 0.1;
      A     DB21.DBX 394.0;
      JNB   M161;
      L     DB21.DBD 206;
      T     MD 588;
      SET;
      SAVE;
      CLR;
M161: A     BR;
      );
      JNB   M162;
      L     DB21.DBD 210;
      T     MD 592;
M162: NOP   0;
      A(;
      A     L 0.1;
      AN    DB21.DBX 394.0;
      JNB   M163;
      L     DB21.DBD 214;
      T     MD 588;
      SET;
      SAVE;
      CLR;
M163: A     BR;
      );
      JNB   M164;
      L     DB21.DBD 218;
      T     MD 592;
M164: NOP   0;
      A     L 0.0;
      A(;
      A(;
      L     DB21.DBW 370;
      L     11;
      ==I;
      );
      A     M 11.4;
      O;
      A     M 11.2;
      A(;
      L     DB7.DBB 375;
      L     12;
      ==I;
      );
      A(;
      O(;
      L     DB7.DBW 2;
      L     5;
      ==I;
      );
      O(;
      L     DB7.DBW 2;
      L     11;
      ==I;
      );
      );
      );
      =     L 0.1;
      A(;
      A     L 0.1;
      A     DB21.DBX 394.0;
      JNB   M165;
      L     DB21.DBD 222;
      T     MD 588;
      SET;
      SAVE;
      CLR;
M165: A     BR;
      );
      JNB   M166;
      L     DB21.DBD 226;
      T     MD 592;
M166: NOP   0;
      A(;
      A     L 0.1;
      AN    DB21.DBX 394.0;
      JNB   M167;
      L     DB21.DBD 230;
      T     MD 588;
      SET;
      SAVE;
      CLR;
M167: A     BR;
      );
      JNB   M168;
      L     DB21.DBD 234;
      T     MD 592;
M168: NOP   0;
      A     L 0.0;
      A(;
      A(;
      L     DB21.DBW 370;
      L     12;
      ==I;
      );
      A     M 11.4;
      O;
      A     M 11.2;
      A(;
      L     DB7.DBB 375;
      L     13;
      ==I;
      );
      A(;
      O(;
      L     DB7.DBW 2;
      L     5;
      ==I;
      );
      O(;
      L     DB7.DBW 2;
      L     11;
      ==I;
      );
      );
      );
      =     L 0.1;
      A(;
      A     L 0.1;
      A     DB21.DBX 394.0;
      JNB   M169;
      L     DB21.DBD 238;
      T     MD 588;
      SET;
      SAVE;
      CLR;
M169: A     BR;
      );
      JNB   M170;
      L     DB21.DBD 242;
      T     MD 592;
M170: NOP   0;
      A(;
      A     L 0.1;
      AN    DB21.DBX 394.0;
      JNB   M171;
      L     DB21.DBD 246;
      T     MD 588;
      SET;
      SAVE;
      CLR;
M171: A     BR;
      );
      JNB   M172;
      L     DB21.DBD 250;
      T     MD 592;
M172: NOP   0;
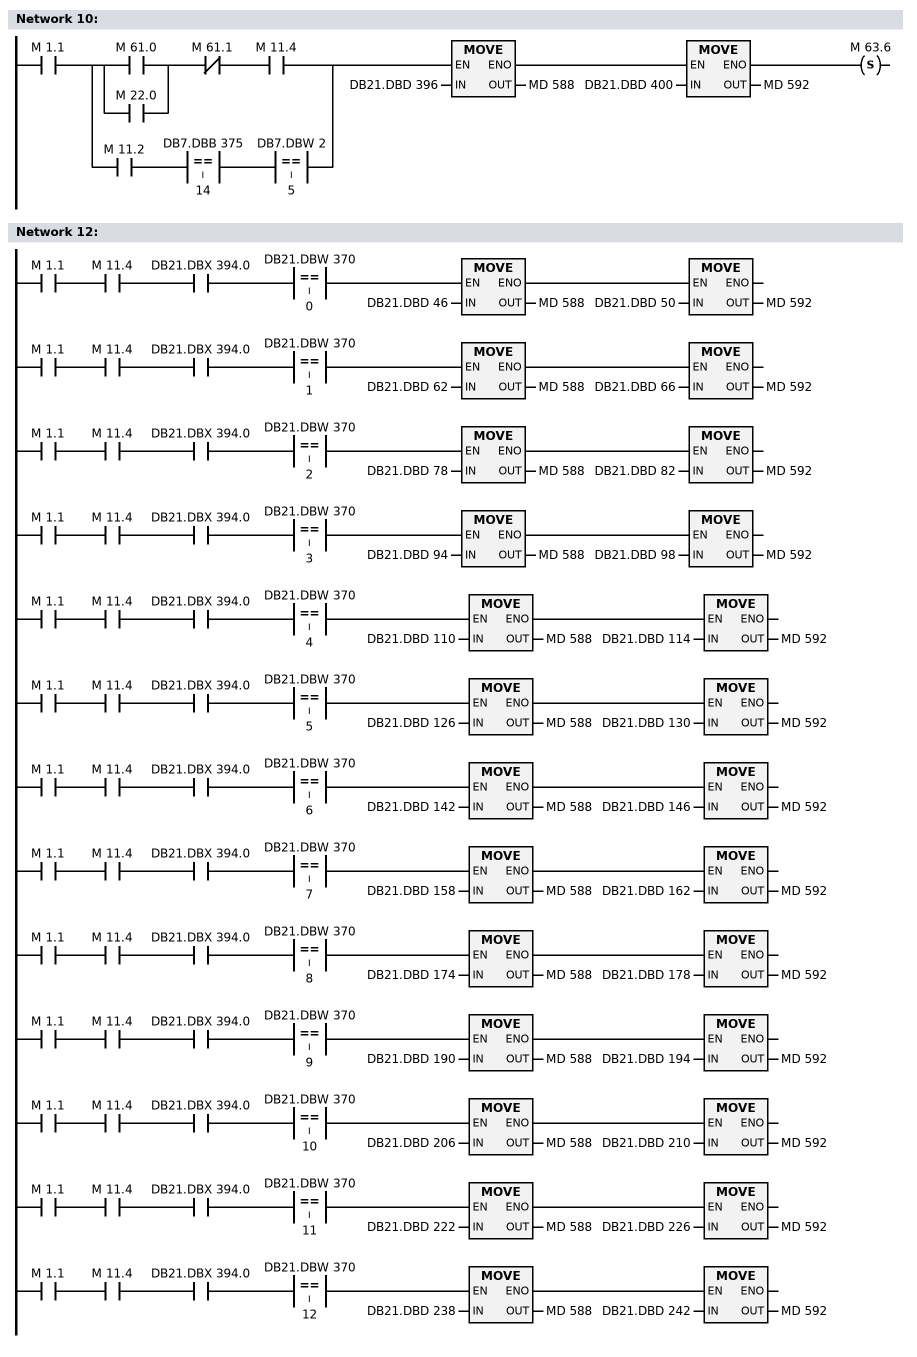
NETWORK
TITLE =
      A(;
      A     M 1.1;
      A(;
      A(;
      O     M 61.0;
      O     M 22.0;
      );
      AN    M 61.1;
      A     M 11.4;
      O;
      A     M 11.2;
      A(;
      L     DB7.DBB 375;
      L     14;
      ==I;
      );
      A(;
      L     DB7.DBW 2;
      L     5;
      ==I;
      );
      );
      JNB   M173;
      L     DB21.DBD 396;
      T     MD 588;
      SET;
      SAVE;
      CLR;
M173: A     BR;
      );
      JNB   M174;
      L     DB21.DBD 400;
      T     MD 592;
      SET;
      SAVE;
      CLR;
M174: A     BR;
      S     M 63.6;
NETWORK
TITLE =
NETWORK
TITLE =
      A     M 1.1;
      A     M 11.4;
      A     DB21.DBX 394.0;
      =     L 0.0;
      A(;
      A     L 0.0;
      A(;
      L     DB21.DBW 370;
      L     0;
      ==I;
      );
      JNB   M175;
      L     DB21.DBD 46;
      T     MD 588;
      SET;
      SAVE;
      CLR;
M175: A     BR;
      );
      JNB   M176;
      L     DB21.DBD 50;
      T     MD 592;
M176: NOP   0;
      A(;
      A     L 0.0;
      A(;
      L     DB21.DBW 370;
      L     1;
      ==I;
      );
      JNB   M177;
      L     DB21.DBD 62;
      T     MD 588;
      SET;
      SAVE;
      CLR;
M177: A     BR;
      );
      JNB   M178;
      L     DB21.DBD 66;
      T     MD 592;
M178: NOP   0;
      A(;
      A     L 0.0;
      A(;
      L     DB21.DBW 370;
      L     2;
      ==I;
      );
      JNB   M179;
      L     DB21.DBD 78;
      T     MD 588;
      SET;
      SAVE;
      CLR;
M179: A     BR;
      );
      JNB   M180;
      L     DB21.DBD 82;
      T     MD 592;
M180: NOP   0;
      A(;
      A     L 0.0;
      A(;
      L     DB21.DBW 370;
      L     3;
      ==I;
      );
      JNB   M181;
      L     DB21.DBD 94;
      T     MD 588;
      SET;
      SAVE;
      CLR;
M181: A     BR;
      );
      JNB   M182;
      L     DB21.DBD 98;
      T     MD 592;
M182: NOP   0;
      A(;
      A     L 0.0;
      A(;
      L     DB21.DBW 370;
      L     4;
      ==I;
      );
      JNB   M183;
      L     DB21.DBD 110;
      T     MD 588;
      SET;
      SAVE;
      CLR;
M183: A     BR;
      );
      JNB   M184;
      L     DB21.DBD 114;
      T     MD 592;
M184: NOP   0;
      A(;
      A     L 0.0;
      A(;
      L     DB21.DBW 370;
      L     5;
      ==I;
      );
      JNB   M185;
      L     DB21.DBD 126;
      T     MD 588;
      SET;
      SAVE;
      CLR;
M185: A     BR;
      );
      JNB   M186;
      L     DB21.DBD 130;
      T     MD 592;
M186: NOP   0;
      A(;
      A     L 0.0;
      A(;
      L     DB21.DBW 370;
      L     6;
      ==I;
      );
      JNB   M187;
      L     DB21.DBD 142;
      T     MD 588;
      SET;
      SAVE;
      CLR;
M187: A     BR;
      );
      JNB   M188;
      L     DB21.DBD 146;
      T     MD 592;
M188: NOP   0;
      A(;
      A     L 0.0;
      A(;
      L     DB21.DBW 370;
      L     7;
      ==I;
      );
      JNB   M189;
      L     DB21.DBD 158;
      T     MD 588;
      SET;
      SAVE;
      CLR;
M189: A     BR;
      );
      JNB   M190;
      L     DB21.DBD 162;
      T     MD 592;
M190: NOP   0;
      A(;
      A     L 0.0;
      A(;
      L     DB21.DBW 370;
      L     8;
      ==I;
      );
      JNB   M191;
      L     DB21.DBD 174;
      T     MD 588;
      SET;
      SAVE;
      CLR;
M191: A     BR;
      );
      JNB   M192;
      L     DB21.DBD 178;
      T     MD 592;
M192: NOP   0;
      A(;
      A     L 0.0;
      A(;
      L     DB21.DBW 370;
      L     9;
      ==I;
      );
      JNB   M193;
      L     DB21.DBD 190;
      T     MD 588;
      SET;
      SAVE;
      CLR;
M193: A     BR;
      );
      JNB   M194;
      L     DB21.DBD 194;
      T     MD 592;
M194: NOP   0;
      A(;
      A     L 0.0;
      A(;
      L     DB21.DBW 370;
      L     10;
      ==I;
      );
      JNB   M195;
      L     DB21.DBD 206;
      T     MD 588;
      SET;
      SAVE;
      CLR;
M195: A     BR;
      );
      JNB   M196;
      L     DB21.DBD 210;
      T     MD 592;
M196: NOP   0;
      A(;
      A     L 0.0;
      A(;
      L     DB21.DBW 370;
      L     11;
      ==I;
      );
      JNB   M197;
      L     DB21.DBD 222;
      T     MD 588;
      SET;
      SAVE;
      CLR;
M197: A     BR;
      );
      JNB   M198;
      L     DB21.DBD 226;
      T     MD 592;
M198: NOP   0;
      A(;
      A     L 0.0;
      A(;
      L     DB21.DBW 370;
      L     12;
      ==I;
      );
      JNB   M199;
      L     DB21.DBD 238;
      T     MD 588;
      SET;
      SAVE;
      CLR;
M199: A     BR;
      );
      JNB   M200;
      L     DB21.DBD 242;
      T     MD 592;
M200: NOP   0;
NETWORK
TITLE =
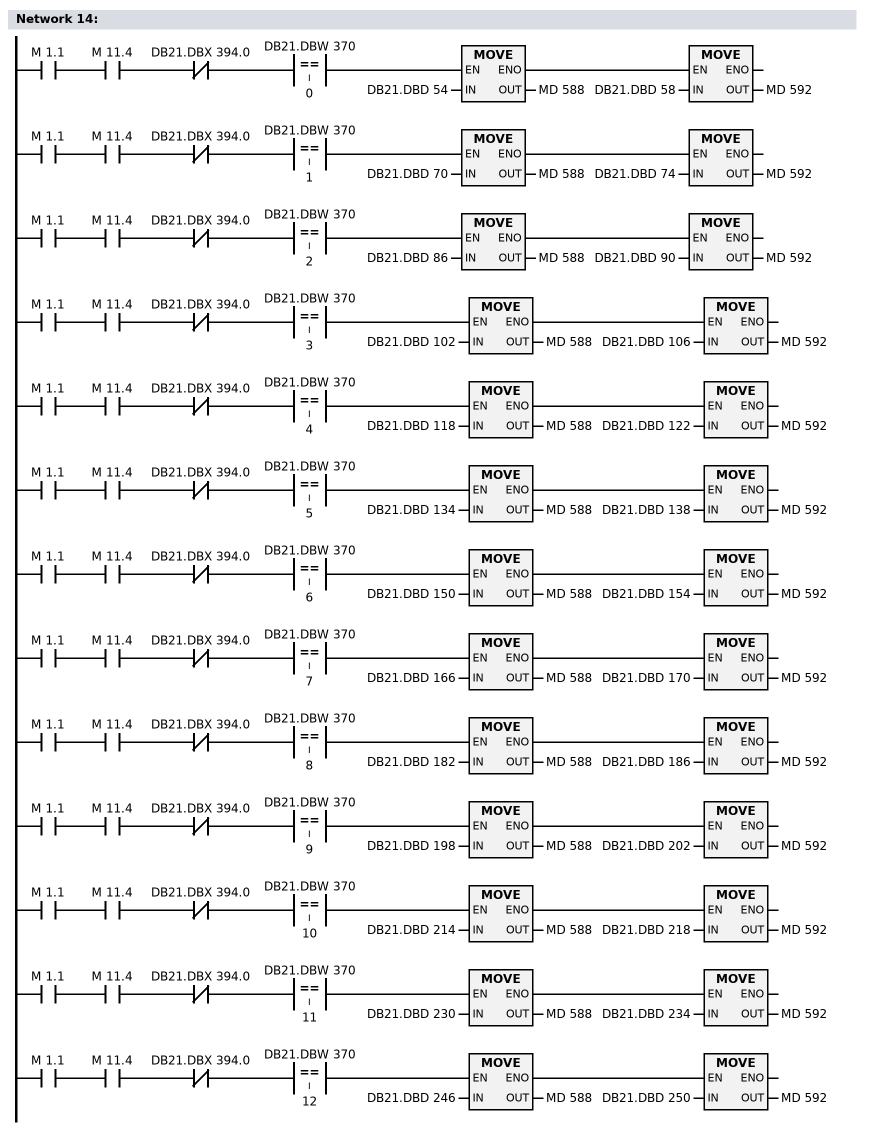
NETWORK
TITLE =
      A     M 1.1;
      A     M 11.4;
      AN    DB21.DBX 394.0;
      =     L 0.0;
      A(;
      A     L 0.0;
      A(;
      L     DB21.DBW 370;
      L     0;
      ==I;
      );
      JNB   M201;
      L     DB21.DBD 54;
      T     MD 588;
      SET;
      SAVE;
      CLR;
M201: A     BR;
      );
      JNB   M202;
      L     DB21.DBD 58;
      T     MD 592;
M202: NOP   0;
      A(;
      A     L 0.0;
      A(;
      L     DB21.DBW 370;
      L     1;
      ==I;
      );
      JNB   M203;
      L     DB21.DBD 70;
      T     MD 588;
      SET;
      SAVE;
      CLR;
M203: A     BR;
      );
      JNB   M204;
      L     DB21.DBD 74;
      T     MD 592;
M204: NOP   0;
      A(;
      A     L 0.0;
      A(;
      L     DB21.DBW 370;
      L     2;
      ==I;
      );
      JNB   M205;
      L     DB21.DBD 86;
      T     MD 588;
      SET;
      SAVE;
      CLR;
M205: A     BR;
      );
      JNB   M206;
      L     DB21.DBD 90;
      T     MD 592;
M206: NOP   0;
      A(;
      A     L 0.0;
      A(;
      L     DB21.DBW 370;
      L     3;
      ==I;
      );
      JNB   M207;
      L     DB21.DBD 102;
      T     MD 588;
      SET;
      SAVE;
      CLR;
M207: A     BR;
      );
      JNB   M208;
      L     DB21.DBD 106;
      T     MD 592;
M208: NOP   0;
      A(;
      A     L 0.0;
      A(;
      L     DB21.DBW 370;
      L     4;
      ==I;
      );
      JNB   M209;
      L     DB21.DBD 118;
      T     MD 588;
      SET;
      SAVE;
      CLR;
M209: A     BR;
      );
      JNB   M210;
      L     DB21.DBD 122;
      T     MD 592;
M210: NOP   0;
      A(;
      A     L 0.0;
      A(;
      L     DB21.DBW 370;
      L     5;
      ==I;
      );
      JNB   M211;
      L     DB21.DBD 134;
      T     MD 588;
      SET;
      SAVE;
      CLR;
M211: A     BR;
      );
      JNB   M212;
      L     DB21.DBD 138;
      T     MD 592;
M212: NOP   0;
      A(;
      A     L 0.0;
      A(;
      L     DB21.DBW 370;
      L     6;
      ==I;
      );
      JNB   M213;
      L     DB21.DBD 150;
      T     MD 588;
      SET;
      SAVE;
      CLR;
M213: A     BR;
      );
      JNB   M214;
      L     DB21.DBD 154;
      T     MD 592;
M214: NOP   0;
      A(;
      A     L 0.0;
      A(;
      L     DB21.DBW 370;
      L     7;
      ==I;
      );
      JNB   M215;
      L     DB21.DBD 166;
      T     MD 588;
      SET;
      SAVE;
      CLR;
M215: A     BR;
      );
      JNB   M216;
      L     DB21.DBD 170;
      T     MD 592;
M216: NOP   0;
      A(;
      A     L 0.0;
      A(;
      L     DB21.DBW 370;
      L     8;
      ==I;
      );
      JNB   M217;
      L     DB21.DBD 182;
      T     MD 588;
      SET;
      SAVE;
      CLR;
M217: A     BR;
      );
      JNB   M218;
      L     DB21.DBD 186;
      T     MD 592;
M218: NOP   0;
      A(;
      A     L 0.0;
      A(;
      L     DB21.DBW 370;
      L     9;
      ==I;
      );
      JNB   M219;
      L     DB21.DBD 198;
      T     MD 588;
      SET;
      SAVE;
      CLR;
M219: A     BR;
      );
      JNB   M220;
      L     DB21.DBD 202;
      T     MD 592;
M220: NOP   0;
      A(;
      A     L 0.0;
      A(;
      L     DB21.DBW 370;
      L     10;
      ==I;
      );
      JNB   M221;
      L     DB21.DBD 214;
      T     MD 588;
      SET;
      SAVE;
      CLR;
M221: A     BR;
      );
      JNB   M222;
      L     DB21.DBD 218;
      T     MD 592;
M222: NOP   0;
      A(;
      A     L 0.0;
      A(;
      L     DB21.DBW 370;
      L     11;
      ==I;
      );
      JNB   M223;
      L     DB21.DBD 230;
      T     MD 588;
      SET;
      SAVE;
      CLR;
M223: A     BR;
      );
      JNB   M224;
      L     DB21.DBD 234;
      T     MD 592;
M224: NOP   0;
      A(;
      A     L 0.0;
      A(;
      L     DB21.DBW 370;
      L     12;
      ==I;
      );
      JNB   M225;
      L     DB21.DBD 246;
      T     MD 588;
      SET;
      SAVE;
      CLR;
M225: A     BR;
      );
      JNB   M226;
      L     DB21.DBD 250;
      T     MD 592;
M226: NOP   0;
NETWORK
TITLE =
END_FUNCTION

FUNCTION FC 81 : VOID
VERSION : 0.1
BEGIN
// (block stored without names or comments; labels and parameter names are numbered)
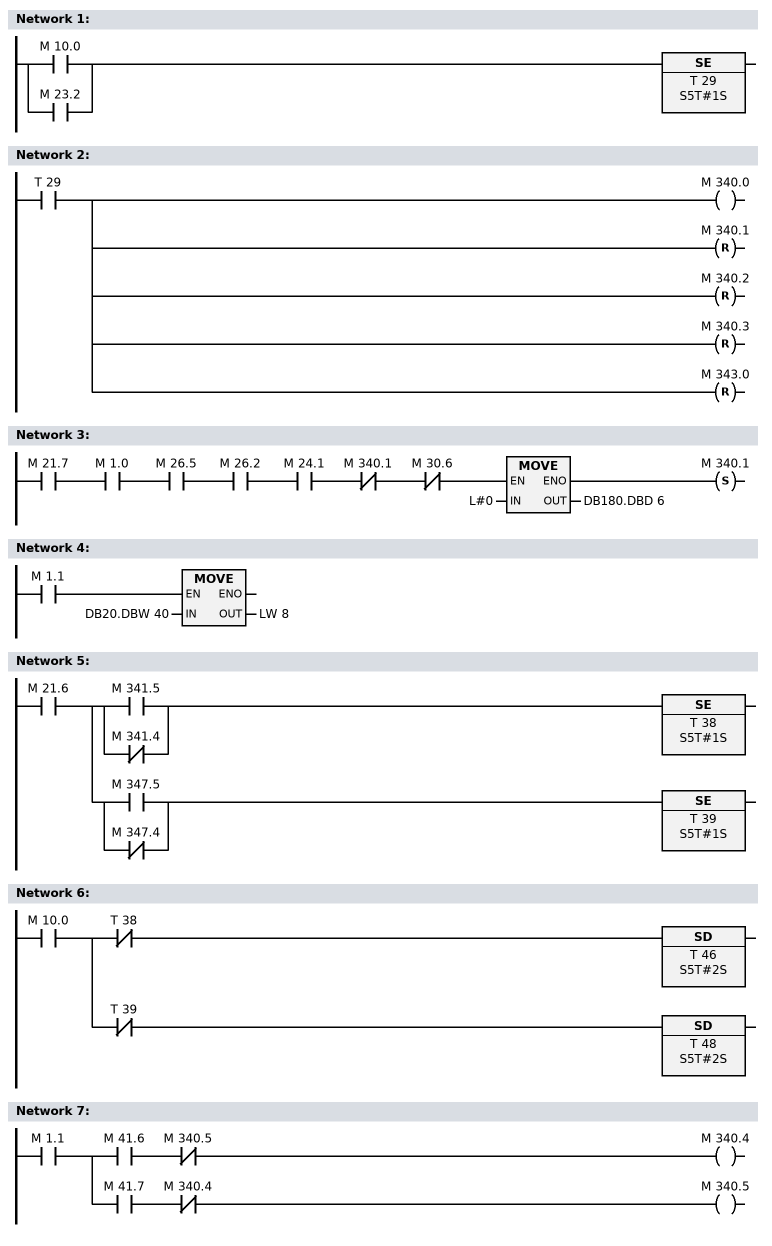
NETWORK
TITLE =
      O     M 10.0;
      O     M 23.2;
      L     S5T#1S;
      SE    T 29;
NETWORK
TITLE =
      A     T 29;
      =     M 340.0;
      R     M 340.1;
      R     M 340.2;
      R     M 340.3;
      R     M 343.0;
NETWORK
TITLE =
      A     M 21.7;
      A     M 1.0;
      A     M 26.5;
      A     M 26.2;
      A     M 24.1;
      AN    M 340.1;
      AN    M 30.6;
      JNB   M001;
      L     L#0;
      T     DB180.DBD 6;
      SET;
      SAVE;
      CLR;
M001: A     BR;
      S     M 340.1;
NETWORK
TITLE =
      A     M 1.1;
      JNB   M002;
      L     DB20.DBW 40;
      T     LW 8;
M002: NOP   0;
NETWORK
TITLE =
      A     M 21.6;
      =     L 15.0;
      A     L 15.0;
      A(;
      O     M 341.5;
      ON    M 341.4;
      );
      L     S5T#1S;
      SE    T 38;
      A     L 15.0;
      A(;
      O     M 347.5;
      ON    M 347.4;
      );
      L     S5T#1S;
      SE    T 39;
NETWORK
TITLE =
      A     M 10.0;
      =     L 15.0;
      A     L 15.0;
      AN    T 38;
      L     S5T#2S;
      SD    T 46;
      A     L 15.0;
      AN    T 39;
      L     S5T#2S;
      SD    T 48;
NETWORK
TITLE =
      A     M 1.1;
      =     L 15.0;
      A     L 15.0;
      A     M 41.6;
      AN    M 340.5;
      =     M 340.4;
      A     L 15.0;
      A     M 41.7;
      AN    M 340.4;
      =     M 340.5;
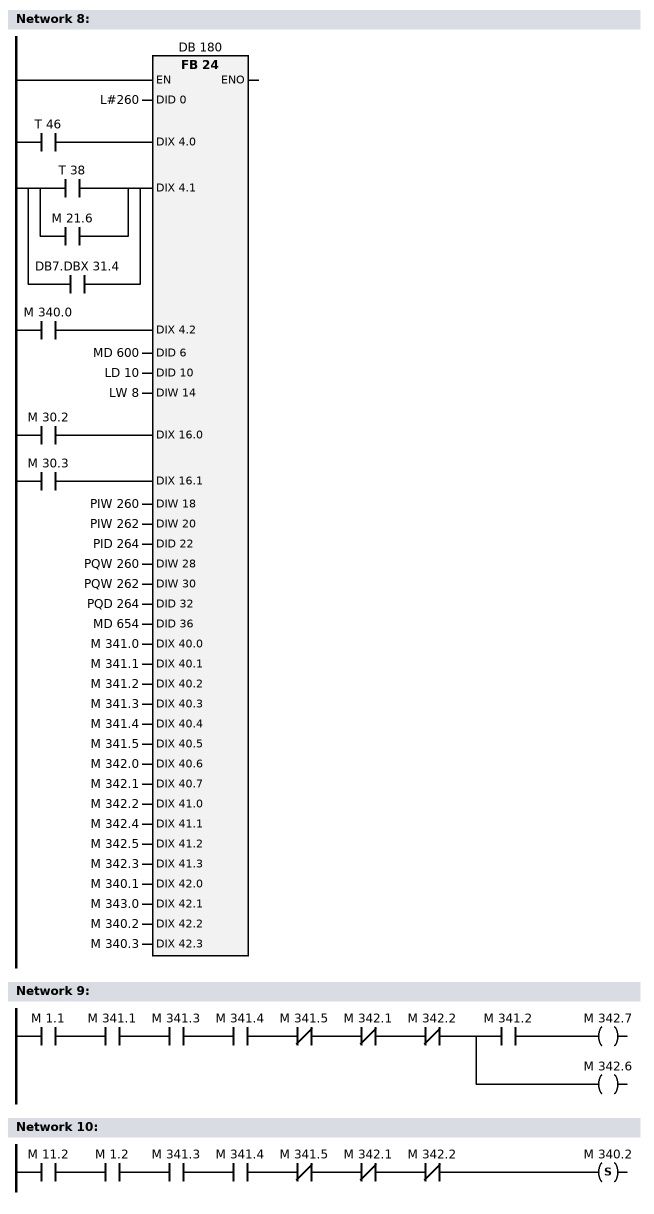
NETWORK
TITLE =
      A     T 46;
      =     L 15.0;
      BLD   103;
      A(;
      O     T 38;
      O     M 21.6;
      O     DB7.DBX 31.4;
      );
      =     L 15.1;
      BLD   103;
      A     M 340.0;
      =     L 15.2;
      BLD   103;
      A     M 30.2;
      =     L 15.3;
      BLD   103;
      A     M 30.3;
      =     L 15.4;
      BLD   103;
      CALL  FB 24 , DB 180 (
           DID 0                    := L#260,
           DIX 4.0                  := L 15.0,
           DIX 4.1                  := L 15.1,
           DIX 4.2                  := L 15.2,
           DID 6                    := MD 600,
           DID 10                   := LD 10,
           DIW 14                   := LW 8,
           DIX 16.0                 := L 15.3,
           DIX 16.1                 := L 15.4,
           DIW 18                   := PIW 260,
           DIW 20                   := PIW 262,
           DID 22                   := PID 264,
           DIW 28                   := PQW 260,
           DIW 30                   := PQW 262,
           DID 32                   := PQD 264,
           DID 36                   := MD 654,
           DIX 40.0                 := M 341.0,
           DIX 40.1                 := M 341.1,
           DIX 40.2                 := M 341.2,
           DIX 40.3                 := M 341.3,
           DIX 40.4                 := M 341.4,
           DIX 40.5                 := M 341.5,
           DIX 40.6                 := M 342.0,
           DIX 40.7                 := M 342.1,
           DIX 41.0                 := M 342.2,
           DIX 41.1                 := M 342.4,
           DIX 41.2                 := M 342.5,
           DIX 41.3                 := M 342.3,
           DIX 42.0                 := M 340.1,
           DIX 42.1                 := M 343.0,
           DIX 42.2                 := M 340.2,
           DIX 42.3                 := M 340.3);
      NOP   0;
NETWORK
TITLE =
      A     M 1.1;
      A     M 341.1;
      A     M 341.3;
      A     M 341.4;
      AN    M 341.5;
      AN    M 342.1;
      AN    M 342.2;
      =     L 15.0;
      A     L 15.0;
      A     M 341.2;
      =     M 342.7;
      A     L 15.0;
      BLD   102;
      =     M 342.6;
NETWORK
TITLE =
      A     M 11.2;
      A     M 1.2;
      A     M 341.3;
      A     M 341.4;
      AN    M 341.5;
      AN    M 342.1;
      AN    M 342.2;
      S     M 340.2;
NETWORK
TITLE =
NETWORK
TITLE =
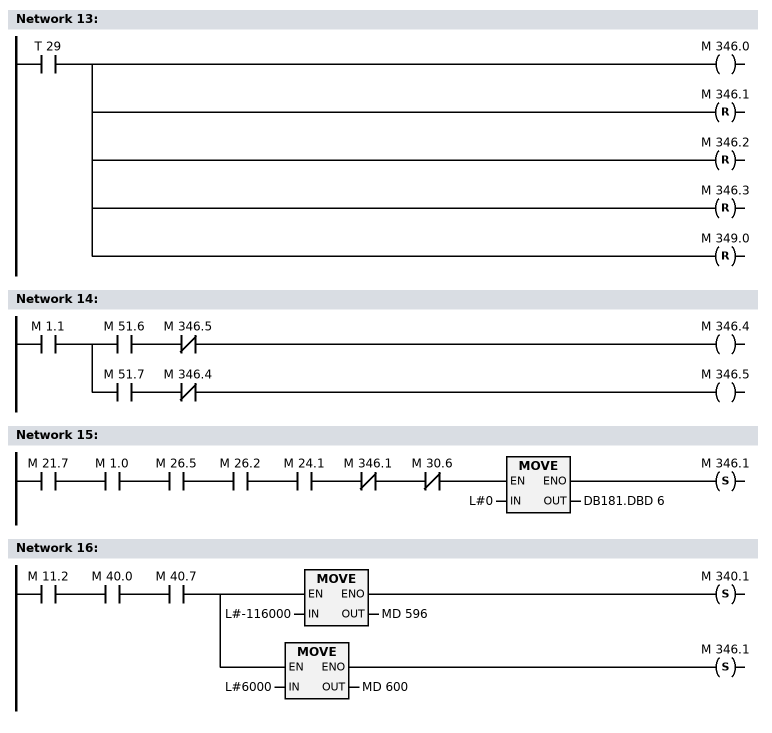
NETWORK
TITLE =
      A     T 29;
      =     M 346.0;
      R     M 346.1;
      R     M 346.2;
      R     M 346.3;
      R     M 349.0;
NETWORK
TITLE =
      A     M 1.1;
      =     L 15.0;
      A     L 15.0;
      A     M 51.6;
      AN    M 346.5;
      =     M 346.4;
      A     L 15.0;
      A     M 51.7;
      AN    M 346.4;
      =     M 346.5;
NETWORK
TITLE =
      A     M 21.7;
      A     M 1.0;
      A     M 26.5;
      A     M 26.2;
      A     M 24.1;
      AN    M 346.1;
      AN    M 30.6;
      JNB   M003;
      L     L#0;
      T     DB181.DBD 6;
      SET;
      SAVE;
      CLR;
M003: A     BR;
      S     M 346.1;
NETWORK
TITLE =
      A     M 11.2;
      A     M 40.0;
      A     M 40.7;
      =     L 15.0;
      A     L 15.0;
      JNB   M004;
      L     L#-116000;
      T     MD 596;
      SET;
      SAVE;
      CLR;
M004: A     BR;
      S     M 340.1;
      A     L 15.0;
      JNB   M005;
      L     L#6000;
      T     MD 600;
      SET;
      SAVE;
      CLR;
M005: A     BR;
      S     M 346.1;
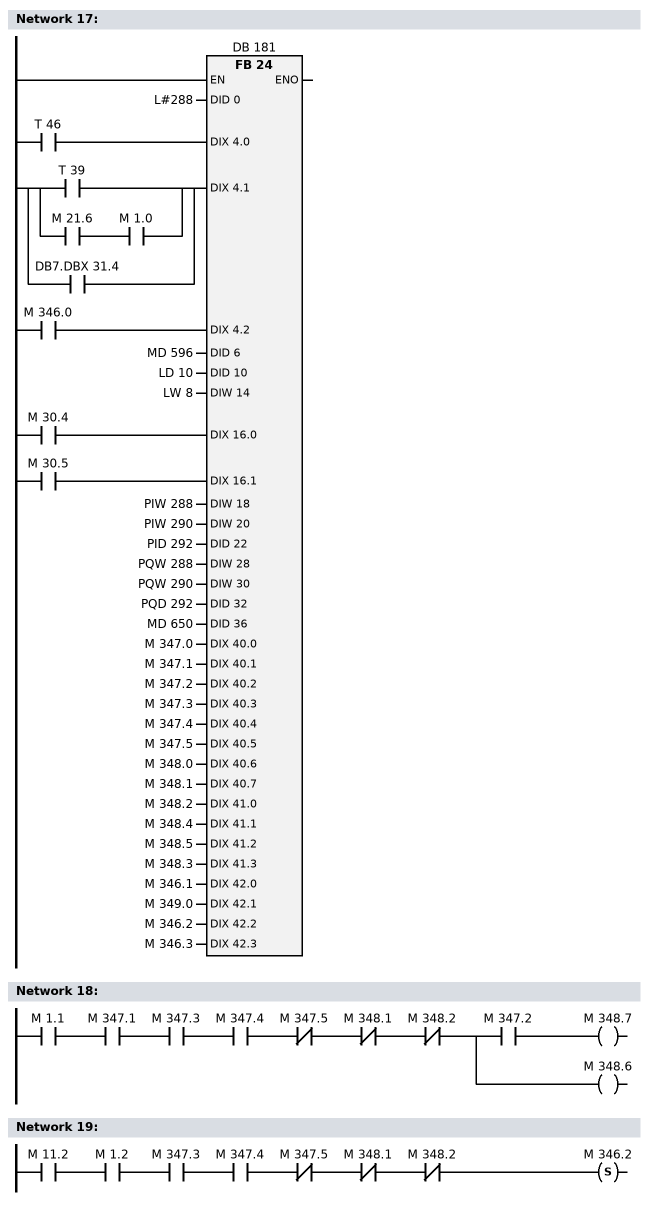
NETWORK
TITLE =
      A     T 46;
      =     L 15.0;
      BLD   103;
      A(;
      O     T 39;
      O;
      A     M 21.6;
      A     M 1.0;
      O     DB7.DBX 31.4;
      );
      =     L 15.1;
      BLD   103;
      A     M 346.0;
      =     L 15.2;
      BLD   103;
      A     M 30.4;
      =     L 15.3;
      BLD   103;
      A     M 30.5;
      =     L 15.4;
      BLD   103;
      CALL  FB 24 , DB 181 (
           DID 0                    := L#288,
           DIX 4.0                  := L 15.0,
           DIX 4.1                  := L 15.1,
           DIX 4.2                  := L 15.2,
           DID 6                    := MD 596,
           DID 10                   := LD 10,
           DIW 14                   := LW 8,
           DIX 16.0                 := L 15.3,
           DIX 16.1                 := L 15.4,
           DIW 18                   := PIW 288,
           DIW 20                   := PIW 290,
           DID 22                   := PID 292,
           DIW 28                   := PQW 288,
           DIW 30                   := PQW 290,
           DID 32                   := PQD 292,
           DID 36                   := MD 650,
           DIX 40.0                 := M 347.0,
           DIX 40.1                 := M 347.1,
           DIX 40.2                 := M 347.2,
           DIX 40.3                 := M 347.3,
           DIX 40.4                 := M 347.4,
           DIX 40.5                 := M 347.5,
           DIX 40.6                 := M 348.0,
           DIX 40.7                 := M 348.1,
           DIX 41.0                 := M 348.2,
           DIX 41.1                 := M 348.4,
           DIX 41.2                 := M 348.5,
           DIX 41.3                 := M 348.3,
           DIX 42.0                 := M 346.1,
           DIX 42.1                 := M 349.0,
           DIX 42.2                 := M 346.2,
           DIX 42.3                 := M 346.3);
      NOP   0;
NETWORK
TITLE =
      A     M 1.1;
      A     M 347.1;
      A     M 347.3;
      A     M 347.4;
      AN    M 347.5;
      AN    M 348.1;
      AN    M 348.2;
      =     L 15.0;
      A     L 15.0;
      A     M 347.2;
      =     M 348.7;
      A     L 15.0;
      BLD   102;
      =     M 348.6;
NETWORK
TITLE =
      A     M 11.2;
      A     M 1.2;
      A     M 347.3;
      A     M 347.4;
      AN    M 347.5;
      AN    M 348.1;
      AN    M 348.2;
      S     M 346.2;
END_FUNCTION

FUNCTION FC 117 : VOID
VERSION : 0.1
BEGIN
// (block stored without names or comments; labels and parameter names are numbered)
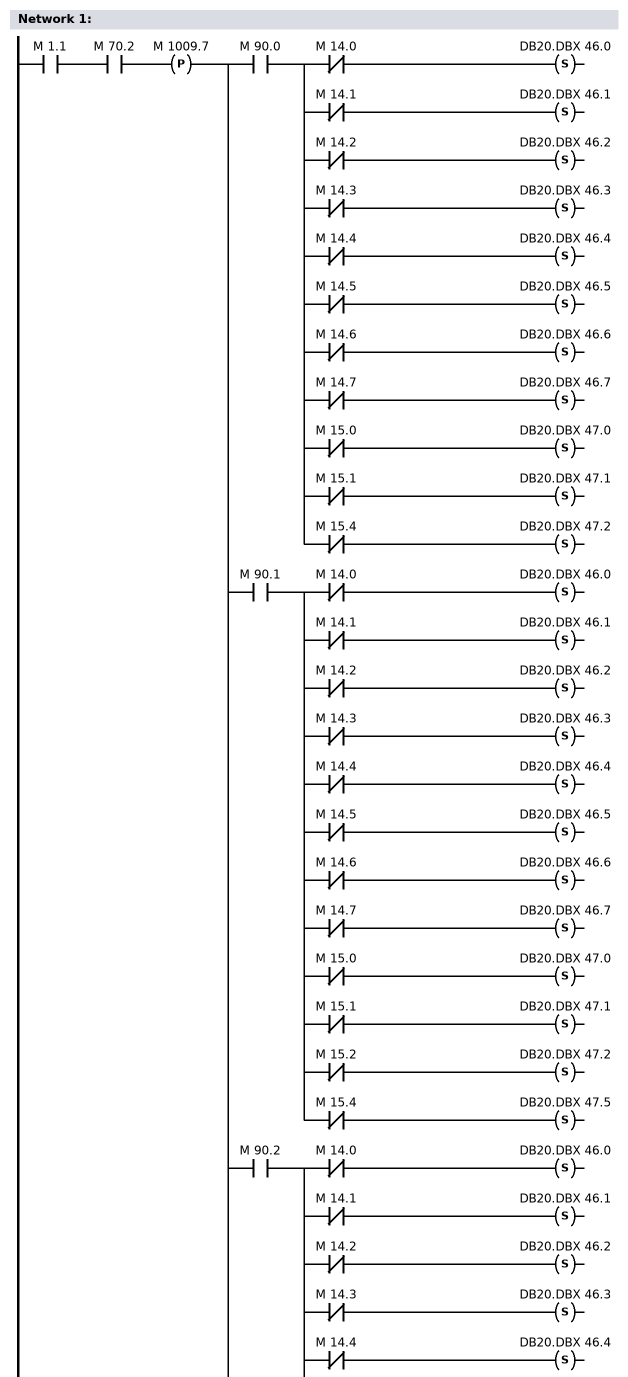
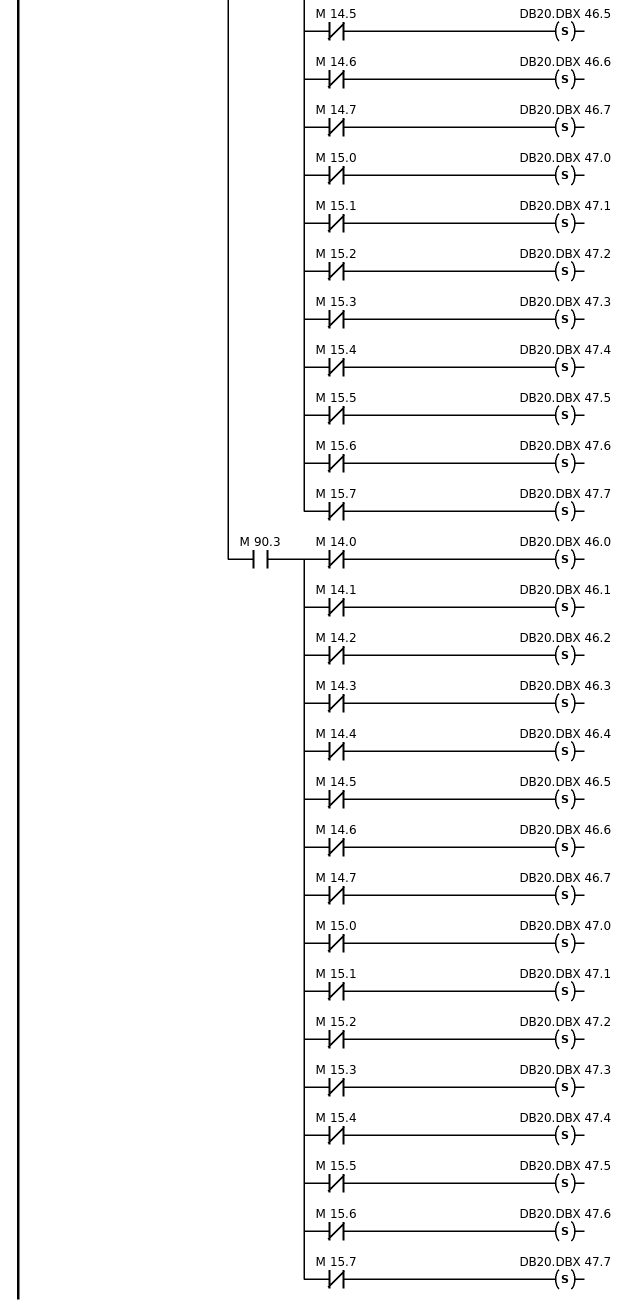
NETWORK
TITLE =
      A     M 1.1;
      A     M 70.2;
      FP    M 1009.7;
      =     L 0.0;
      A     L 0.0;
      A     M 90.0;
      =     L 0.1;
      A     L 0.1;
      AN    M 14.0;
      S     DB20.DBX 46.0;
      A     L 0.1;
      AN    M 14.1;
      S     DB20.DBX 46.1;
      A     L 0.1;
      AN    M 14.2;
      S     DB20.DBX 46.2;
      A     L 0.1;
      AN    M 14.3;
      S     DB20.DBX 46.3;
      A     L 0.1;
      AN    M 14.4;
      S     DB20.DBX 46.4;
      A     L 0.1;
      AN    M 14.5;
      S     DB20.DBX 46.5;
      A     L 0.1;
      AN    M 14.6;
      S     DB20.DBX 46.6;
      A     L 0.1;
      AN    M 14.7;
      S     DB20.DBX 46.7;
      A     L 0.1;
      AN    M 15.0;
      S     DB20.DBX 47.0;
      A     L 0.1;
      AN    M 15.1;
      S     DB20.DBX 47.1;
      A     L 0.1;
      AN    M 15.4;
      S     DB20.DBX 47.2;
      A     L 0.0;
      A     M 90.1;
      =     L 0.1;
      A     L 0.1;
      AN    M 14.0;
      S     DB20.DBX 46.0;
      A     L 0.1;
      AN    M 14.1;
      S     DB20.DBX 46.1;
      A     L 0.1;
      AN    M 14.2;
      S     DB20.DBX 46.2;
      A     L 0.1;
      AN    M 14.3;
      S     DB20.DBX 46.3;
      A     L 0.1;
      AN    M 14.4;
      S     DB20.DBX 46.4;
      A     L 0.1;
      AN    M 14.5;
      S     DB20.DBX 46.5;
      A     L 0.1;
      AN    M 14.6;
      S     DB20.DBX 46.6;
      A     L 0.1;
      AN    M 14.7;
      S     DB20.DBX 46.7;
      A     L 0.1;
      AN    M 15.0;
      S     DB20.DBX 47.0;
      A     L 0.1;
      AN    M 15.1;
      S     DB20.DBX 47.1;
      A     L 0.1;
      AN    M 15.2;
      S     DB20.DBX 47.2;
      A     L 0.1;
      AN    M 15.4;
      S     DB20.DBX 47.5;
      A     L 0.0;
      A     M 90.2;
      =     L 0.1;
      A     L 0.1;
      AN    M 14.0;
      S     DB20.DBX 46.0;
      A     L 0.1;
      AN    M 14.1;
      S     DB20.DBX 46.1;
      A     L 0.1;
      AN    M 14.2;
      S     DB20.DBX 46.2;
      A     L 0.1;
      AN    M 14.3;
      S     DB20.DBX 46.3;
      A     L 0.1;
      AN    M 14.4;
      S     DB20.DBX 46.4;
      A     L 0.1;
      AN    M 14.5;
      S     DB20.DBX 46.5;
      A     L 0.1;
      AN    M 14.6;
      S     DB20.DBX 46.6;
      A     L 0.1;
      AN    M 14.7;
      S     DB20.DBX 46.7;
      A     L 0.1;
      AN    M 15.0;
      S     DB20.DBX 47.0;
      A     L 0.1;
      AN    M 15.1;
      S     DB20.DBX 47.1;
      A     L 0.1;
      AN    M 15.2;
      S     DB20.DBX 47.2;
      A     L 0.1;
      AN    M 15.3;
      S     DB20.DBX 47.3;
      A     L 0.1;
      AN    M 15.4;
      S     DB20.DBX 47.4;
      A     L 0.1;
      AN    M 15.5;
      S     DB20.DBX 47.5;
      A     L 0.1;
      AN    M 15.6;
      S     DB20.DBX 47.6;
      A     L 0.1;
      AN    M 15.7;
      S     DB20.DBX 47.7;
      A     L 0.0;
      A     M 90.3;
      =     L 0.1;
      A     L 0.1;
      AN    M 14.0;
      S     DB20.DBX 46.0;
      A     L 0.1;
      AN    M 14.1;
      S     DB20.DBX 46.1;
      A     L 0.1;
      AN    M 14.2;
      S     DB20.DBX 46.2;
      A     L 0.1;
      AN    M 14.3;
      S     DB20.DBX 46.3;
      A     L 0.1;
      AN    M 14.4;
      S     DB20.DBX 46.4;
      A     L 0.1;
      AN    M 14.5;
      S     DB20.DBX 46.5;
      A     L 0.1;
      AN    M 14.6;
      S     DB20.DBX 46.6;
      A     L 0.1;
      AN    M 14.7;
      S     DB20.DBX 46.7;
      A     L 0.1;
      AN    M 15.0;
      S     DB20.DBX 47.0;
      A     L 0.1;
      AN    M 15.1;
      S     DB20.DBX 47.1;
      A     L 0.1;
      AN    M 15.2;
      S     DB20.DBX 47.2;
      A     L 0.1;
      AN    M 15.3;
      S     DB20.DBX 47.3;
      A     L 0.1;
      AN    M 15.4;
      S     DB20.DBX 47.4;
      A     L 0.1;
      AN    M 15.5;
      S     DB20.DBX 47.5;
      A     L 0.1;
      AN    M 15.6;
      S     DB20.DBX 47.6;
      A     L 0.1;
      AN    M 15.7;
      S     DB20.DBX 47.7;
END_FUNCTION

FUNCTION FC 800 : VOID
AUTHOR : Cellini
FAMILY : GCLib
NAME : TimeOut
VERSION : 1.0
BEGIN
// (block stored without names or comments; labels and parameter names are numbered)
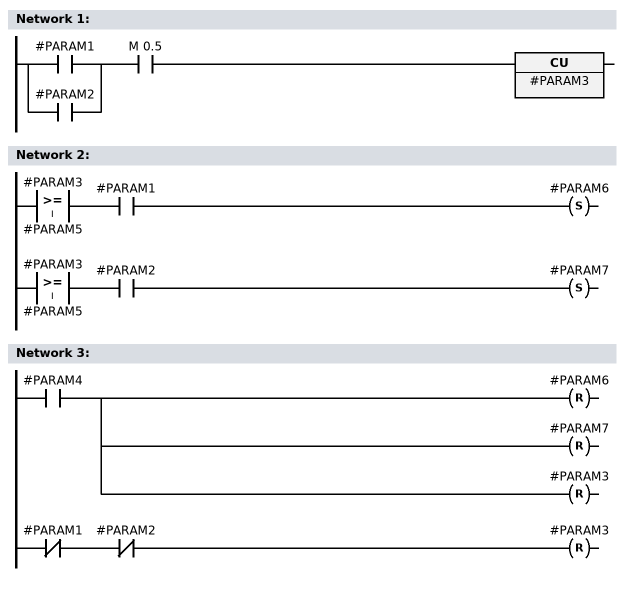
NETWORK
TITLE =
      A     #PARAM1;
      O     #PARAM2;
      A     M 0.5;
      CU    #PARAM3;
NETWORK
TITLE =
      L     #PARAM3;
      L     #PARAM5;
      >=I;
      A     #PARAM1;
      S     #PARAM6;
      L     #PARAM3;
      L     #PARAM5;
      >=I;
      A     #PARAM2;
      S     #PARAM7;
NETWORK
TITLE =
      A     #PARAM4;
      R     #PARAM6;
      R     #PARAM7;
      R     #PARAM3;
      AN    #PARAM1;
      AN    #PARAM2;
      R     #PARAM3;
END_FUNCTION

DATA_BLOCK DB 5
AUTHOR : Salvati
VERSION : 0.0
FB 20
BEGIN
END_DATA_BLOCK

DATA_BLOCK DB 7
AUTHOR : Coletti
FAMILY : GCLib
VERSION : 0.1
BEGIN
// 382 bytes; values not shown
END_DATA_BLOCK

DATA_BLOCK DB 11
VERSION : 0.1
BEGIN
// 38 bytes; values not shown
END_DATA_BLOCK

DATA_BLOCK DB 12
VERSION : 0.1
BEGIN
// 38 bytes; values not shown
END_DATA_BLOCK

DATA_BLOCK DB 13
VERSION : 0.1
BEGIN
// 16 bytes; values not shown
END_DATA_BLOCK

DATA_BLOCK DB 20
VERSION : 0.1
BEGIN
// 72 bytes; values not shown
END_DATA_BLOCK

DATA_BLOCK DB 21
AUTHOR : Coletti
VERSION : 0.1
BEGIN
// 478 bytes; values not shown
END_DATA_BLOCK

DATA_BLOCK DB 22
VERSION : 0.1
BEGIN
// 8860 bytes; values not shown
END_DATA_BLOCK

DATA_BLOCK DB 23
VERSION : 0.1
BEGIN
// 2 bytes; values not shown
END_DATA_BLOCK

DATA_BLOCK DB 180
VERSION : 0.0
FB 24
BEGIN
END_DATA_BLOCK

DATA_BLOCK DB 181
VERSION : 0.0
FB 24
BEGIN
END_DATA_BLOCK

ORGANIZATION_BLOCK OB 1
VERSION : 0.1
BEGIN
// (block stored without names or comments; labels and parameter names are numbered)
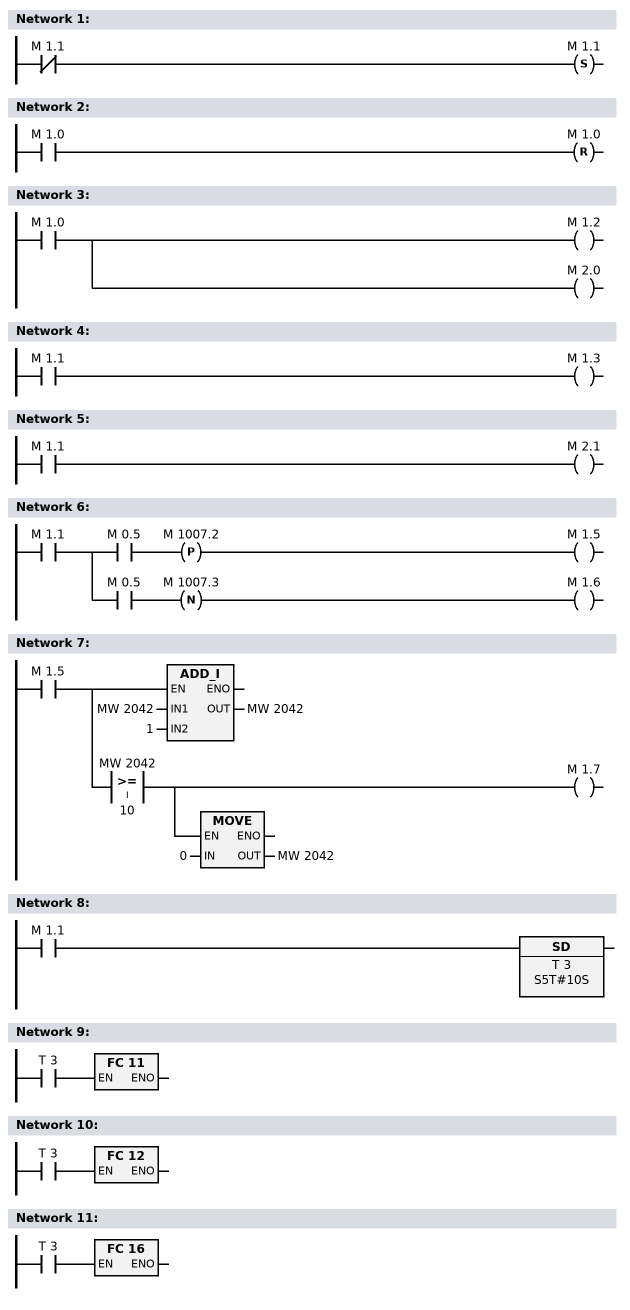
NETWORK
TITLE =
      AN    M 1.1;
      S     M 1.1;
NETWORK
TITLE =
      A     M 1.0;
      R     M 1.0;
NETWORK
TITLE =
      A     M 1.0;
      =     M 1.2;
      =     M 2.0;
NETWORK
TITLE =
      A     M 1.1;
      =     M 1.3;
NETWORK
TITLE =
      A     M 1.1;
      =     M 2.1;
NETWORK
TITLE =
      A     M 1.1;
      =     L 20.0;
      A     L 20.0;
      A     M 0.5;
      FP    M 1007.2;
      =     M 1.5;
      A     L 20.0;
      A     M 0.5;
      FN    M 1007.3;
      =     M 1.6;
NETWORK
TITLE =
      A     M 1.5;
      =     L 20.0;
      A     L 20.0;
      JNB   M001;
      L     MW 2042;
      L     1;
      +I;
      T     MW 2042;
M001: NOP   0;
      A     L 20.0;
      A(;
      L     MW 2042;
      L     10;
      >=I;
      );
      =     L 20.1;
      A     L 20.1;
      BLD   102;
      =     M 1.7;
      A     L 20.1;
      JNB   M002;
      L     0;
      T     MW 2042;
M002: NOP   0;
NETWORK
TITLE =
      A     M 1.1;
      L     S5T#10S;
      SD    T 3;
NETWORK
TITLE =
      A     T 3;
      JNB   M003;
      CALL  FC 11;
M003: NOP   0;
NETWORK
TITLE =
      A     T 3;
      JNB   M004;
      CALL  FC 12;
M004: NOP   0;
NETWORK
TITLE =
      A     T 3;
      JNB   M005;
      CALL  FC 16;
M005: NOP   0;
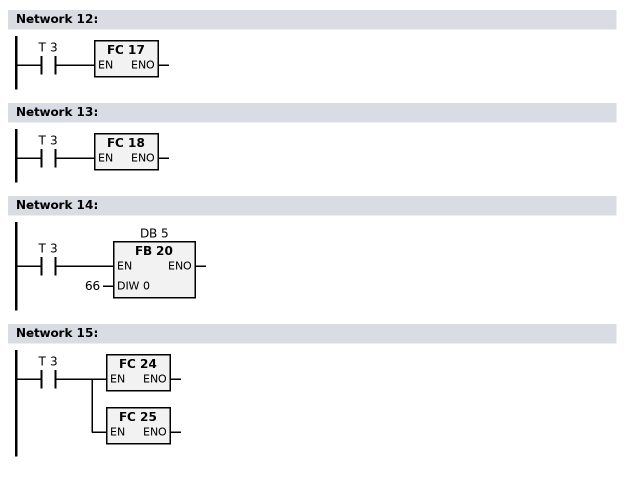
NETWORK
TITLE =
      A     T 3;
      JNB   M006;
      CALL  FC 17;
M006: NOP   0;
NETWORK
TITLE =
      A     T 3;
      JNB   M007;
      CALL  FC 18;
M007: NOP   0;
NETWORK
TITLE =
      A     T 3;
      JNB   M008;
      CALL  FB 20 , DB 5 (
           DIW 0                    := 66);
M008: NOP   0;
NETWORK
TITLE =
      A     T 3;
      =     L 20.0;
      A     L 20.0;
      JNB   M009;
      CALL  FC 24;
M009: NOP   0;
      A     L 20.0;
      JNB   M010;
      CALL  FC 25;
M010: NOP   0;
END_ORGANIZATION_BLOCK

ORGANIZATION_BLOCK OB 82
VERSION : 1.0
BEGIN
// (block stored without names or comments; labels and parameter names are numbered)
NETWORK
TITLE =
END_ORGANIZATION_BLOCK

ORGANIZATION_BLOCK OB 86
VERSION : 0.1
BEGIN
// (block stored without names or comments; labels and parameter names are numbered)
NETWORK
TITLE =
END_ORGANIZATION_BLOCK

ORGANIZATION_BLOCK OB 100
VERSION : 0.1
BEGIN
// (block stored without names or comments; labels and parameter names are numbered)
